LIN {X 0,Y 425.301,Z 259.752,A -85,B 0,C 180,E1 15177.061,E2 15177.061} C_VEL
LIN {X 0,Y 425.303,Z 259.751,A -85,B 0,C 180,E1 15173.169,E2 15173.169} C_VEL
LIN {X 0,Y 425.314,Z 259.743,A -85,B 0,C 180,E1 15169.371,E2 15169.371} C_VEL
LIN {X 0,Y 425.315,Z 259.738,A -85,B 0,C 180,E1 15165.531,E2 15165.531} C_VEL
LIN {X 0,Y 425.318,Z 259.739,A -85,B 0,C 180,E1 15161.623,E2 15161.623} C_VEL
LIN {X 0,Y 425.32,Z 259.754,A -85,B 0,C 180,E1 15157.829,E2 15157.829} C_VEL
LIN {X 0,Y 425.32,Z 259.751,A -85,B 0,C 180,E1 15153.921,E2 15153.921} C_VEL
LIN {X 0,Y 425.319,Z 259.736,A -85,B 0,C 180,E1 15150.046,E2 15150.046} C_VEL
LIN {X 0,Y 425.304,Z 259.744,A -85,B 0,C 180,E1 15146.228,E2 15146.228} C_VEL
LIN {X 0,Y 425.298,Z 259.757,A -85,B 0,C 180,E1 15142.385,E2 15142.385} C_VEL
LIN {X 0,Y 425.297,Z 259.743,A -85,B 0,C 180,E1 15138.503,E2 15138.503} C_VEL
LIN {X 0,Y 425.3,Z 259.734,A -85,B 0,C 180,E1 15134.707,E2 15134.707} C_VEL
LIN {X 0,Y 425.309,Z 259.756,A -85,B 0,C 180,E1 15130.839,E2 15130.839} C_VEL
LIN {X 0,Y 425.321,Z 259.742,A -85,B 0,C 180,E1 15127.02,E2 15127.02} C_VEL
LIN {X 0,Y 425.315,Z 259.735,A -85,B 0,C 180,E1 15123.098,E2 15123.098} C_VEL
LIN {X 0,Y 425.324,Z 259.753,A -85,B 0,C 180,E1 15119.325,E2 15119.325} C_VEL
LIN {X 0,Y 425.313,Z 259.752,A -85,B 0,C 180,E1 15115.414,E2 15115.414} C_VEL
LIN {X 0,Y 425.303,Z 259.742,A -85,B 0,C 180,E1 15111.618,E2 15111.618} C_VEL
LIN {X 0,Y 425.292,Z 259.736,A -85,B 0,C 180,E1 15107.784,E2 15107.784} C_VEL
LIN {X 0,Y 425.293,Z 259.748,A -85,B 0,C 180,E1 15104.033,E2 15104.033} C_VEL
LIN {X 0,Y 425.3,Z 259.753,A -85,B 0,C 180,E1 15100.211,E2 15100.211} C_VEL
LIN {X 0,Y 425.317,Z 259.755,A -85,B 0,C 180,E1 15096.443,E2 15096.443} C_VEL
LIN {X 0,Y 425.321,Z 259.752,A -85,B 0,C 180,E1 15092.563,E2 15092.563} C_VEL
LIN {X 0,Y 425.323,Z 259.747,A -85,B 0,C 180,E1 15088.698,E2 15088.698} C_VEL
LIN {X 0,Y 425.316,Z 259.743,A -85,B 0,C 180,E1 15084.832,E2 15084.832} C_VEL
LIN {X 0,Y 425.328,Z 259.912,A -85,B 0,C 180,E1 15083.057,E2 15083.057} C_VEL
LIN {X 0,Y 426.138,Z 262.4,A -85,B 0,C 180,E1 15082.576,E2 15082.576} C_VEL
LIN {X 0,Y 427.707,Z 264.913,A -85,B 0,C 180,E1 15082.061,E2 15082.061} C_VEL
LIN {X 0,Y 435.111,Z 279.75,A -85,B 0,C 180,E1 15079.434,E2 15079.434} C_VEL
LIN {X 0,Y 442.483,Z 295.067,A -85,B 0,C 180,E1 15076.967,E2 15076.967} C_VEL
LIN {X 0,Y 445.89,Z 302.403,A -85,B 0,C 180,E1 15075.916,E2 15075.916} C_VEL
LIN {X 0,Y 457.017,Z 320.95,A -85,B 0,C 180,E1 15074.239,E2 15074.239} C_VEL
LIN {X 0,Y 458.902,Z 336.106,A -85,B 0,C 180,E1 15073.722,E2 15073.722} C_VEL
LIN {X 0,Y 453.344,Z 551.105,A -85,B 0,C 180,E1 15070.004,E2 15070.004} C_VEL
LIN {X 0,Y 451.835,Z 606.521,A -85,B 0,C 180,E1 15069.024,E2 15069.024} C_VEL
LIN {X 0,Y 450.386,Z 628.482,A -85,B 0,C 180,E1 15068.425,E2 15068.425} C_VEL
LIN {X 0,Y 448.608,Z 649.294,A -85,B 0,C 180,E1 15067.637,E2 15067.637} C_VEL
LIN {X 0,Y 446.489,Z 669.88,A -85,B 0,C 180,E1 15066.638,E2 15066.638} C_VEL
LIN {X 0,Y 444.025,Z 690.18,A -85,B 0,C 180,E1 15065.397,E2 15065.397} C_VEL
LIN {X 0,Y 441.401,Z 709.749,A -85,B 0,C 180,E1 15063.941,E2 15063.941} C_VEL
LIN {X 0,Y 438.704,Z 728.638,A -85,B 0,C 180,E1 15062.268,E2 15062.268} C_VEL
LIN {X 0,Y 436.021,Z 746.682,A -85,B 0,C 180,E1 15060.372,E2 15060.372} C_VEL
LIN {X 0,Y 433.442,Z 763.445,A -85,B 0,C 180,E1 15058.295,E2 15058.295} C_VEL
LIN {X 0,Y 430.954,Z 780.217,A -85,B 0,C 180,E1 15055.858,E2 15055.858} C_VEL
LIN {X 0,Y 428.999,Z 794.198,A -85,B 0,C 180,E1 15053.485,E2 15053.485} C_VEL
LIN {X 0,Y 427.355,Z 806.771,A -85,B 0,C 180,E1 15050.974,E2 15050.974} C_VEL
LIN {X 0,Y 426.058,Z 818.033,A -85,B 0,C 180,E1 15048.327,E2 15048.327} C_VEL
LIN {X 0,Y 425.11,Z 827.973,A -85,B 0,C 180,E1 15045.551,E2 15045.551} C_VEL
LIN {X 0,Y 424.495,Z 835.991,A -85,B 0,C 180,E1 15042.79,E2 15042.79} C_VEL
LIN {X 0,Y 424.136,Z 842.606,A -85,B 0,C 180,E1 15039.908,E2 15039.908} C_VEL
LIN {X 0,Y 423.986,Z 847.351,A -85,B 0,C 180,E1 15037.178,E2 15037.178} C_VEL
LIN {X 0,Y 423.92,Z 850.446,A -85,B 0,C 180,E1 15034.463,E2 15034.463} C_VEL
LIN {X 0,Y 423.9,Z 852.175,A -85,B 0,C 180,E1 15031.756,E2 15031.756} C_VEL
LIN {X 0,Y 423.907,Z 852.32,A -85,B 0,C 180,E1 15029.053,E2 15029.053} C_VEL
LIN {X 0,Y 423.91,Z 851.039,A -85,B 0,C 180,E1 15026.212,E2 15026.212} C_VEL
LIN {X 0,Y 423.947,Z 848.381,A -85,B 0,C 180,E1 15023.634,E2 15023.634} C_VEL
LIN {X 0,Y 424.084,Z 843.921,A -85,B 0,C 180,E1 15020.773,E2 15020.773} C_VEL
LIN {X 0,Y 424.358,Z 838.352,A -85,B 0,C 180,E1 15018.17,E2 15018.17} C_VEL
LIN {X 0,Y 424.886,Z 830.435,A -85,B 0,C 180,E1 15015.276,E2 15015.276} C_VEL
LIN {X 0,Y 425.726,Z 821.114,A -85,B 0,C 180,E1 15012.504,E2 15012.504} C_VEL
LIN {X 0,Y 426.894,Z 810.324,A -85,B 0,C 180,E1 15009.86,E2 15009.86} C_VEL
LIN {X 0,Y 428.488,Z 797.377,A -85,B 0,C 180,E1 15007.179,E2 15007.179} C_VEL
LIN {X 0,Y 430.418,Z 783.285,A -85,B 0,C 180,E1 15004.694,E2 15004.694} C_VEL
LIN {X 0,Y 432.668,Z 767.834,A -85,B 0,C 180,E1 15002.369,E2 15002.369} C_VEL
LIN {X 0,Y 435.112,Z 751.206,A -85,B 0,C 180,E1 15000.24,E2 15000.24} C_VEL
LIN {X 0,Y 437.827,Z 732.887,A -85,B 0,C 180,E1 14998.237,E2 14998.237} C_VEL
LIN {X 0,Y 440.485,Z 714.446,A -85,B 0,C 180,E1 14996.523,E2 14996.523} C_VEL
LIN {X 0,Y 443.086,Z 695.133,A -85,B 0,C 180,E1 14995.027,E2 14995.027} C_VEL
LIN {X 0,Y 445.497,Z 675.185,A -85,B 0,C 180,E1 14993.743,E2 14993.743} C_VEL
LIN {X 0,Y 447.751,Z 654.688,A -85,B 0,C 180,E1 14992.67,E2 14992.67} C_VEL
LIN {X 0,Y 449.597,Z 634.166,A -85,B 0,C 180,E1 14991.836,E2 14991.836} C_VEL
LIN {X 0,Y 451.161,Z 611.946,A -85,B 0,C 180,E1 14991.172,E2 14991.172} C_VEL
LIN {X 0,Y 452.131,Z 587.924,A -85,B 0,C 180,E1 14990.684,E2 14990.684} C_VEL
LIN {X 0,Y 457.639,Z 367.78,A -85,B 0,C 180,E1 14986.894,E2 14986.894} C_VEL
LIN {X 0,Y 458.383,Z 333.61,A -85,B 0,C 180,E1 14986.271,E2 14986.271} C_VEL
LIN {X 0,Y 456.385,Z 319.925,A -85,B 0,C 180,E1 14985.758,E2 14985.758} C_VEL
LIN {X 0,Y 445.461,Z 301.473,A -85,B 0,C 180,E1 14984.048,E2 14984.048} C_VEL
LIN {X 0,Y 438.428,Z 285.88,A -85,B 0,C 180,E1 14981.579,E2 14981.579} C_VEL
LIN {X 0,Y 432.266,Z 273.434,A -85,B 0,C 180,E1 14979.33,E2 14979.33} C_VEL
LIN {X 0,Y 429.39,Z 268.237,A -85,B 0,C 180,E1 14978.273,E2 14978.273} C_VEL
LIN {X 0,Y 427.403,Z 264.222,A -85,B 0,C 180,E1 14977.463,E2 14977.463} C_VEL
LIN {X 0,Y 425.54,Z 260.917,A -85,B 0,C 180,E1 14976.726,E2 14976.726} C_VEL
LIN {X 0,Y 425.313,Z 259.812,A -85,B 0,C 180,E1 14976.395,E2 14976.395} C_VEL
LIN {X 0,Y 425.308,Z 259.758,A -85,B 0,C 180,E1 14972.573,E2 14972.573} C_VEL
LIN {X 0,Y 425.315,Z 259.748,A -85,B 0,C 180,E1 14968.731,E2 14968.731} C_VEL
LIN {X 0,Y 425.317,Z 259.757,A -85,B 0,C 180,E1 14964.846,E2 14964.846} C_VEL
LIN {X 0,Y 425.314,Z 259.749,A -85,B 0,C 180,E1 14961.043,E2 14961.043} C_VEL
LIN {X 0,Y 425.303,Z 259.747,A -85,B 0,C 180,E1 14957.231,E2 14957.231} C_VEL
LIN {X 0,Y 425.3,Z 259.753,A -85,B 0,C 180,E1 14953.46,E2 14953.46} C_VEL
LIN {X 0,Y 425.301,Z 259.76,A -85,B 0,C 180,E1 14949.61,E2 14949.61} C_VEL
LIN {X 0,Y 425.309,Z 259.756,A -85,B 0,C 180,E1 14945.803,E2 14945.803} C_VEL
LIN {X 0,Y 425.317,Z 259.749,A -85,B 0,C 180,E1 14942.022,E2 14942.022} C_VEL
LIN {X 0,Y 425.32,Z 259.746,A -85,B 0,C 180,E1 14938.25,E2 14938.25} C_VEL
LIN {X 0,Y 425.317,Z 259.756,A -85,B 0,C 180,E1 14934.335,E2 14934.335} C_VEL
LIN {X 0,Y 425.29,Z 259.754,A -85,B 0,C 180,E1 14930.666,E2 14930.666} C_VEL
LIN {X 0,Y 425.273,Z 259.761,A -85,B 0,C 180,E1 14926.957,E2 14926.957} C_VEL
LIN {X 0,Y 425.297,Z 259.923,A -85,B 0,C 180,E1 14924.805,E2 14924.805} C_VEL
LIN {X 0,Y 426.13,Z 262.406,A -85,B 0,C 180,E1 14924.207,E2 14924.207} C_VEL
LIN {X 0,Y 427.697,Z 265.015,A -85,B 0,C 180,E1 14923.57,E2 14923.57} C_VEL
LIN {X 0,Y 432.042,Z 273.926,A -85,B 0,C 180,E1 14921.656,E2 14921.656} C_VEL
LIN {X 0,Y 438.633,Z 288.164,A -85,B 0,C 180,E1 14918.892,E2 14918.892} C_VEL
LIN {X 0,Y 443.787,Z 300.497,A -85,B 0,C 180,E1 14916.798,E2 14916.798} C_VEL
LIN {X 0,Y 453.343,Z 316.481,A -85,B 0,C 180,E1 14915.244,E2 14915.244} C_VEL
LIN {X 0,Y 455.959,Z 333.247,A -85,B 0,C 180,E1 14914.568,E2 14914.568} C_VEL
LIN {X 0,Y 448.532,Z 567.509,A -85,B 0,C 180,E1 14910.326,E2 14910.326} C_VEL
LIN {X 0,Y 447.276,Z 588.491,A -85,B 0,C 180,E1 14909.711,E2 14909.711} C_VEL
LIN {X 0,Y 445.669,Z 608.284,A -85,B 0,C 180,E1 14908.896,E2 14908.896} C_VEL
LIN {X 0,Y 443.645,Z 628.289,A -85,B 0,C 180,E1 14907.823,E2 14907.823} C_VEL
LIN {X 0,Y 441.394,Z 647.121,A -85,B 0,C 180,E1 14906.553,E2 14906.553} C_VEL
LIN {X 0,Y 439.116,Z 664.26,A -85,B 0,C 180,E1 14905.146,E2 14905.146} C_VEL
LIN {X 0,Y 436.553,Z 681.806,A -85,B 0,C 180,E1 14903.408,E2 14903.408} C_VEL
LIN {X 0,Y 434.022,Z 698.14,A -85,B 0,C 180,E1 14901.455,E2 14901.455} C_VEL
LIN {X 0,Y 431.753,Z 712.503,A -85,B 0,C 180,E1 14899.405,E2 14899.405} C_VEL
LIN {X 0,Y 429.664,Z 725.853,A -85,B 0,C 180,E1 14897.142,E2 14897.142} C_VEL
LIN {X 0,Y 427.831,Z 738.286,A -85,B 0,C 180,E1 14894.611,E2 14894.611} C_VEL
LIN {X 0,Y 427.439,Z 741.15,A -85,B 0,C 180,E1 14893.967,E2 14893.967} C_VEL
LIN {X 0,Y 425.985,Z 745.086,A -85,B 0,C 180,E1 14893.089,E2 14893.089} C_VEL
LIN {X 0,Y 419.031,Z 754.446,A -85,B 0,C 180,E1 14890.859,E2 14890.859} C_VEL
LIN {X 0,Y 417.682,Z 757.489,A -85,B 0,C 180,E1 14889.897,E2 14889.897} C_VEL
LIN {X 0,Y 416.881,Z 764.999,A -85,B 0,C 180,E1 14886.999,E2 14886.999} C_VEL
LIN {X 0,Y 416.439,Z 770.435,A -85,B 0,C 180,E1 14884.184,E2 14884.184} C_VEL
LIN {X 0,Y 416.212,Z 774.156,A -85,B 0,C 180,E1 14881.42,E2 14881.42} C_VEL
LIN {X 0,Y 416.135,Z 776.403,A -85,B 0,C 180,E1 14878.565,E2 14878.565} C_VEL
LIN {X 0,Y 416.109,Z 777.068,A -85,B 0,C 180,E1 14875.782,E2 14875.782} C_VEL
LIN {X 0,Y 416.131,Z 776.179,A -85,B 0,C 180,E1 14873.042,E2 14873.042} C_VEL
LIN {X 0,Y 416.214,Z 773.712,A -85,B 0,C 180,E1 14870.24,E2 14870.24} C_VEL
LIN {X 0,Y 416.448,Z 769.461,A -85,B 0,C 180,E1 14867.322,E2 14867.322} C_VEL
LIN {X 0,Y 416.897,Z 763.841,A -85,B 0,C 180,E1 14864.587,E2 14864.587} C_VEL
LIN {X 0,Y 417.65,Z 756.615,A -85,B 0,C 180,E1 14861.883,E2 14861.883} C_VEL
LIN {X 0,Y 418.842,Z 747.081,A -85,B 0,C 180,E1 14859.066,E2 14859.066} C_VEL
LIN {X 0,Y 420.424,Z 735.997,A -85,B 0,C 180,E1 14856.419,E2 14856.419} C_VEL
LIN {X 0,Y 422.248,Z 724.149,A -85,B 0,C 180,E1 14854.075,E2 14854.075} C_VEL
LIN {X 0,Y 424.353,Z 711.065,A -85,B 0,C 180,E1 14851.892,E2 14851.892} C_VEL
LIN {X 0,Y 426.769,Z 696.203,A -85,B 0,C 180,E1 14849.8,E2 14849.8} C_VEL
LIN {X 0,Y 429.265,Z 680.441,A -85,B 0,C 180,E1 14847.932,E2 14847.932} C_VEL
LIN {X 0,Y 431.865,Z 663.081,A -85,B 0,C 180,E1 14846.217,E2 14846.217} C_VEL
LIN {X 0,Y 434.365,Z 644.633,A -85,B 0,C 180,E1 14844.718,E2 14844.718} C_VEL
LIN {X 0,Y 436.594,Z 626.086,A -85,B 0,C 180,E1 14843.492,E2 14843.492} C_VEL
LIN {X 0,Y 438.597,Z 606.057,A -85,B 0,C 180,E1 14842.436,E2 14842.436} C_VEL
LIN {X 0,Y 440.289,Z 585.271,A -85,B 0,C 180,E1 14841.612,E2 14841.612} C_VEL
LIN {X 0,Y 441.466,Z 564.974,A -85,B 0,C 180,E1 14841.039,E2 14841.039} C_VEL
LIN {X 0,Y 448.439,Z 333.3,A -85,B 0,C 180,E1 14836.885,E2 14836.885} C_VEL
LIN {X 0,Y 445.796,Z 318.48,A -85,B 0,C 180,E1 14836.272,E2 14836.272} C_VEL
LIN {X 0,Y 434.687,Z 299.71,A -85,B 0,C 180,E1 14834.524,E2 14834.524} C_VEL
LIN {X 0,Y 427.785,Z 283.545,A -85,B 0,C 180,E1 14831.75,E2 14831.75} C_VEL
LIN {X 0,Y 422.474,Z 272.072,A -85,B 0,C 180,E1 14829.581,E2 14829.581} C_VEL
LIN {X 0,Y 419.084,Z 264.754,A -85,B 0,C 180,E1 14828.133,E2 14828.133} C_VEL
LIN {X 0,Y 417.393,Z 260.937,A -85,B 0,C 180,E1 14827.316,E2 14827.316} C_VEL
LIN {X 0,Y 417.378,Z 260.734,A -85,B 0,C 180,E1 14823.848,E2 14823.848} C_VEL
LIN {X 0,Y 417.382,Z 260.747,A -85,B 0,C 180,E1 14819.958,E2 14819.958} C_VEL
LIN {X 0,Y 417.38,Z 260.747,A -85,B 0,C 180,E1 14815.979,E2 14815.979} C_VEL
LIN {X 0,Y 417.382,Z 260.746,A -85,B 0,C 180,E1 14812.003,E2 14812.003} C_VEL
LIN {X 0,Y 417.381,Z 260.744,A -85,B 0,C 180,E1 14808.062,E2 14808.062} C_VEL
LIN {X 0,Y 417.379,Z 260.74,A -85,B 0,C 180,E1 14804.193,E2 14804.193} C_VEL
LIN {X 0,Y 417.374,Z 260.727,A -85,B 0,C 180,E1 14800.299,E2 14800.299} C_VEL
LIN {X 0,Y 417.362,Z 260.725,A -85,B 0,C 180,E1 14796.448,E2 14796.448} C_VEL
LIN {X 0,Y 417.36,Z 260.741,A -85,B 0,C 180,E1 14792.615,E2 14792.615} C_VEL
LIN {X 0,Y 417.362,Z 260.745,A -85,B 0,C 180,E1 14788.744,E2 14788.744} C_VEL
LIN {X 0,Y 417.366,Z 260.724,A -85,B 0,C 180,E1 14784.936,E2 14784.936} C_VEL
LIN {X 0,Y 417.376,Z 260.733,A -85,B 0,C 180,E1 14781.058,E2 14781.058} C_VEL
LIN {X 0,Y 417.377,Z 260.744,A -85,B 0,C 180,E1 14777.099,E2 14777.099} C_VEL
LIN {X 0,Y 417.379,Z 260.719,A -85,B 0,C 180,E1 14773.294,E2 14773.294} C_VEL
LIN {X 0,Y 417.379,Z 260.728,A -85,B 0,C 180,E1 14769.374,E2 14769.374} C_VEL
LIN {X 0,Y 417.379,Z 260.744,A -85,B 0,C 180,E1 14765.497,E2 14765.497} C_VEL
LIN {X 0,Y 417.372,Z 260.734,A -85,B 0,C 180,E1 14761.646,E2 14761.646} C_VEL
LIN {X 0,Y 417.355,Z 260.724,A -85,B 0,C 180,E1 14757.94,E2 14757.94} C_VEL
LIN {X 0,Y 417.353,Z 260.741,A -85,B 0,C 180,E1 14754.086,E2 14754.086} C_VEL
LIN {X 0,Y 417.357,Z 260.747,A -85,B 0,C 180,E1 14750.206,E2 14750.206} C_VEL
LIN {X 0,Y 417.368,Z 260.733,A -85,B 0,C 180,E1 14746.421,E2 14746.421} C_VEL
LIN {X 0,Y 417.374,Z 260.728,A -85,B 0,C 180,E1 14742.575,E2 14742.575} C_VEL
LIN {X 0,Y 417.384,Z 260.727,A -85,B 0,C 180,E1 14738.646,E2 14738.646} C_VEL
LIN {X 0,Y 417.38,Z 260.729,A -85,B 0,C 180,E1 14734.759,E2 14734.759} C_VEL
LIN {X 0,Y 417.382,Z 260.729,A -85,B 0,C 180,E1 14730.902,E2 14730.902} C_VEL
LIN {X 0,Y 417.371,Z 260.738,A -85,B 0,C 180,E1 14727.056,E2 14727.056} C_VEL
LIN {X 0,Y 417.408,Z 261.004,A -85,B 0,C 180,E1 14724.197,E2 14724.197} C_VEL
LIN {X 0,Y 418.758,Z 264.378,A -85,B 0,C 180,E1 14723.52,E2 14723.52} C_VEL
LIN {X 0,Y 419.926,Z 266.204,A -85,B 0,C 180,E1 14723.128,E2 14723.128} C_VEL
LIN {X 0,Y 426.82,Z 279.835,A -85,B 0,C 180,E1 14720.591,E2 14720.591} C_VEL
LIN {X 0,Y 434.436,Z 295.417,A -85,B 0,C 180,E1 14717.952,E2 14717.952} C_VEL
LIN {X 0,Y 437.761,Z 302.391,A -85,B 0,C 180,E1 14716.904,E2 14716.904} C_VEL
LIN {X 0,Y 450.827,Z 323.776,A -85,B 0,C 180,E1 14714.879,E2 14714.879} C_VEL
LIN {X 0,Y 451.465,Z 325.832,A -85,B 0,C 180,E1 14714.762,E2 14714.762} C_VEL
LIN {X 0,Y 452.833,Z 337.546,A -85,B 0,C 180,E1 14714.362,E2 14714.362} C_VEL
LIN {X 0,Y 446.973,Z 551.29,A -85,B 0,C 180,E1 14710.621,E2 14710.621} C_VEL
LIN {X 0,Y 445.404,Z 606.186,A -85,B 0,C 180,E1 14709.639,E2 14709.639} C_VEL
LIN {X 0,Y 443.876,Z 628.267,A -85,B 0,C 180,E1 14709.032,E2 14709.032} C_VEL
LIN {X 0,Y 441.975,Z 649.397,A -85,B 0,C 180,E1 14708.221,E2 14708.221} C_VEL
LIN {X 0,Y 439.756,Z 669.844,A -85,B 0,C 180,E1 14707.212,E2 14707.212} C_VEL
LIN {X 0,Y 437.228,Z 689.56,A -85,B 0,C 180,E1 14705.992,E2 14705.992} C_VEL
LIN {X 0,Y 434.471,Z 709.083,A -85,B 0,C 180,E1 14704.525,E2 14704.525} C_VEL
LIN {X 0,Y 431.62,Z 728.067,A -85,B 0,C 180,E1 14702.822,E2 14702.822} C_VEL
LIN {X 0,Y 428.809,Z 745.853,A -85,B 0,C 180,E1 14700.93,E2 14700.93} C_VEL
LIN {X 0,Y 426.062,Z 762.77,A -85,B 0,C 180,E1 14698.806,E2 14698.806} C_VEL
LIN {X 0,Y 423.441,Z 779.408,A -85,B 0,C 180,E1 14696.352,E2 14696.352} C_VEL
LIN {X 0,Y 421.351,Z 793.415,A -85,B 0,C 180,E1 14693.938,E2 14693.938} C_VEL
LIN {X 0,Y 419.527,Z 806.506,A -85,B 0,C 180,E1 14691.271,E2 14691.271} C_VEL
LIN {X 0,Y 418.14,Z 817.819,A -85,B 0,C 180,E1 14688.542,E2 14688.542} C_VEL
LIN {X 0,Y 417.148,Z 827.661,A -85,B 0,C 180,E1 14685.713,E2 14685.713} C_VEL
LIN {X 0,Y 416.521,Z 835.522,A -85,B 0,C 180,E1 14682.939,E2 14682.939} C_VEL
LIN {X 0,Y 416.161,Z 841.887,A -85,B 0,C 180,E1 14680.1,E2 14680.1} C_VEL
LIN {X 0,Y 416.001,Z 846.635,A -85,B 0,C 180,E1 14677.317,E2 14677.317} C_VEL
LIN {X 0,Y 415.946,Z 849.737,A -85,B 0,C 180,E1 14674.548,E2 14674.548} C_VEL
LIN {X 0,Y 415.929,Z 851.481,A -85,B 0,C 180,E1 14671.789,E2 14671.789} C_VEL
LIN {X 0,Y 415.938,Z 851.63,A -85,B 0,C 180,E1 14669.034,E2 14669.034} C_VEL
LIN {X 0,Y 415.938,Z 850.315,A -85,B 0,C 180,E1 14666.139,E2 14666.139} C_VEL
LIN {X 0,Y 415.97,Z 847.646,A -85,B 0,C 180,E1 14663.512,E2 14663.512} C_VEL
LIN {X 0,Y 416.112,Z 843.169,A -85,B 0,C 180,E1 14660.595,E2 14660.595} C_VEL
LIN {X 0,Y 416.393,Z 837.583,A -85,B 0,C 180,E1 14657.94,E2 14657.94} C_VEL
LIN {X 0,Y 416.955,Z 829.643,A -85,B 0,C 180,E1 14654.989,E2 14654.989} C_VEL
LIN {X 0,Y 417.85,Z 820.294,A -85,B 0,C 180,E1 14652.163,E2 14652.163} C_VEL
LIN {X 0,Y 419.089,Z 809.483,A -85,B 0,C 180,E1 14649.468,E2 14649.468} C_VEL
LIN {X 0,Y 420.774,Z 796.654,A -85,B 0,C 180,E1 14646.767,E2 14646.767} C_VEL
LIN {X 0,Y 422.773,Z 782.932,A -85,B 0,C 180,E1 14644.299,E2 14644.299} C_VEL
LIN {X 0,Y 425.145,Z 767.555,A -85,B 0,C 180,E1 14641.941,E2 14641.941} C_VEL
LIN {X 0,Y 427.673,Z 751.38,A -85,B 0,C 180,E1 14639.823,E2 14639.823} C_VEL
LIN {X 0,Y 430.524,Z 733.225,A -85,B 0,C 180,E1 14637.791,E2 14637.791} C_VEL
LIN {X 0,Y 433.317,Z 714.948,A -85,B 0,C 180,E1 14636.053,E2 14636.053} C_VEL
LIN {X 0,Y 436.043,Z 695.823,A -85,B 0,C 180,E1 14634.539,E2 14634.539} C_VEL
LIN {X 0,Y 438.714,Z 675.069,A -85,B 0,C 180,E1 14633.172,E2 14633.172} C_VEL
LIN {X 0,Y 441.125,Z 654.322,A -85,B 0,C 180,E1 14632.072,E2 14632.072} C_VEL
LIN {X 0,Y 443.069,Z 633.728,A -85,B 0,C 180,E1 14631.227,E2 14631.227} C_VEL
LIN {X 0,Y 444.705,Z 611.527,A -85,B 0,C 180,E1 14630.556,E2 14630.556} C_VEL
LIN {X 0,Y 445.729,Z 587.428,A -85,B 0,C 180,E1 14630.062,E2 14630.062} C_VEL
LIN {X 0,Y 451.614,Z 367.128,A -85,B 0,C 180,E1 14626.218,E2 14626.218} C_VEL
LIN {X 0,Y 452.376,Z 335.05,A -85,B 0,C 180,E1 14625.623,E2 14625.623} C_VEL
LIN {X 0,Y 450.779,Z 323.87,A -85,B 0,C 180,E1 14625.195,E2 14625.195} C_VEL
LIN {X 0,Y 439.766,Z 305.361,A -85,B 0,C 180,E1 14623.432,E2 14623.432} C_VEL
LIN {X 0,Y 437.248,Z 301.106,A -85,B 0,C 180,E1 14622.957,E2 14622.957} C_VEL
LIN {X 0,Y 430.638,Z 286.826,A -85,B 0,C 180,E1 14620.55,E2 14620.55} C_VEL
LIN {X 0,Y 424.299,Z 274.319,A -85,B 0,C 180,E1 14618.127,E2 14618.127} C_VEL
LIN {X 0,Y 421.933,Z 269.831,A -85,B 0,C 180,E1 14617.177,E2 14617.177} C_VEL
LIN {X 0,Y 419.29,Z 265.018,A -85,B 0,C 180,E1 14616.087,E2 14616.087} C_VEL
LIN {X 0,Y 417.597,Z 261.86,A -85,B 0,C 180,E1 14615.349,E2 14615.349} C_VEL
LIN {X 0,Y 417.383,Z 260.784,A -85,B 0,C 180,E1 14614.986,E2 14614.986} C_VEL
LIN {X 0,Y 417.38,Z 260.739,A -85,B 0,C 180,E1 14611.161,E2 14611.161} C_VEL
LIN {X 0,Y 417.376,Z 260.742,A -85,B 0,C 180,E1 14607.23,E2 14607.23} C_VEL
LIN {X 0,Y 417.37,Z 260.736,A -85,B 0,C 180,E1 14603.431,E2 14603.431} C_VEL
LIN {X 0,Y 417.369,Z 260.742,A -85,B 0,C 180,E1 14599.597,E2 14599.597} C_VEL
LIN {X 0,Y 417.37,Z 260.747,A -85,B 0,C 180,E1 14595.707,E2 14595.707} C_VEL
LIN {X 0,Y 417.373,Z 260.739,A -85,B 0,C 180,E1 14591.89,E2 14591.89} C_VEL
LIN {X 0,Y 417.382,Z 260.734,A -85,B 0,C 180,E1 14587.988,E2 14587.988} C_VEL
LIN {X 0,Y 417.377,Z 260.735,A -85,B 0,C 180,E1 14584.122,E2 14584.122} C_VEL
LIN {X 0,Y 417.386,Z 260.742,A -85,B 0,C 180,E1 14580.276,E2 14580.276} C_VEL
LIN {X 0,Y 417.373,Z 260.743,A -85,B 0,C 180,E1 14576.43,E2 14576.43} C_VEL
LIN {X 0,Y 417.36,Z 260.738,A -85,B 0,C 180,E1 14572.568,E2 14572.568} C_VEL
LIN {X 0,Y 417.343,Z 260.75,A -85,B 0,C 180,E1 14568.812,E2 14568.812} C_VEL
LIN {X 0,Y 417.418,Z 261.002,A -85,B 0,C 180,E1 14566.142,E2 14566.142} C_VEL
LIN {X 0,Y 419.005,Z 264.731,A -85,B 0,C 180,E1 14565.208,E2 14565.208} C_VEL
LIN {X 0,Y 419.923,Z 266.22,A -85,B 0,C 180,E1 14564.818,E2 14564.818} C_VEL
LIN {X 0,Y 422.649,Z 271.937,A -85,B 0,C 180,E1 14563.509,E2 14563.509} C_VEL
LIN {X 0,Y 426.19,Z 278.883,A -85,B 0,C 180,E1 14561.962,E2 14561.962} C_VEL
LIN {X 0,Y 432.656,Z 293.106,A -85,B 0,C 180,E1 14559.153,E2 14559.153} C_VEL
LIN {X 0,Y 435.89,Z 300.619,A -85,B 0,C 180,E1 14557.851,E2 14557.851} C_VEL
LIN {X 0,Y 446.307,Z 317.854,A -85,B 0,C 180,E1 14556.064,E2 14556.064} C_VEL
LIN {X 0,Y 447.954,Z 321.052,A -85,B 0,C 180,E1 14555.788,E2 14555.788} C_VEL
LIN {X 0,Y 450.008,Z 334.928,A -85,B 0,C 180,E1 14555.226,E2 14555.226} C_VEL
LIN {X 0,Y 442.171,Z 567.894,A -85,B 0,C 180,E1 14550.949,E2 14550.949} C_VEL
LIN {X 0,Y 440.859,Z 588.788,A -85,B 0,C 180,E1 14550.329,E2 14550.329} C_VEL
LIN {X 0,Y 439.239,Z 607.795,A -85,B 0,C 180,E1 14549.544,E2 14549.544} C_VEL
LIN {X 0,Y 437.088,Z 628.269,A -85,B 0,C 180,E1 14548.443,E2 14548.443} C_VEL
LIN {X 0,Y 434.784,Z 646.724,A -85,B 0,C 180,E1 14547.197,E2 14547.197} C_VEL
LIN {X 0,Y 432.374,Z 664.01,A -85,B 0,C 180,E1 14545.776,E2 14545.776} C_VEL
LIN {X 0,Y 429.72,Z 681.134,A -85,B 0,C 180,E1 14544.07,E2 14544.07} C_VEL
LIN {X 0,Y 427.258,Z 696.202,A -85,B 0,C 180,E1 14542.279,E2 14542.279} C_VEL
LIN {X 0,Y 424.701,Z 711.448,A -85,B 0,C 180,E1 14540.13,E2 14540.13} C_VEL
LIN {X 0,Y 422.406,Z 725.223,A -85,B 0,C 180,E1 14537.809,E2 14537.809} C_VEL
LIN {X 0,Y 420.548,Z 736.884,A -85,B 0,C 180,E1 14535.466,E2 14535.466} C_VEL
LIN {X 0,Y 418.957,Z 747.652,A -85,B 0,C 180,E1 14532.858,E2 14532.858} C_VEL
LIN {X 0,Y 417.72,Z 757.152,A -85,B 0,C 180,E1 14530.011,E2 14530.011} C_VEL
LIN {X 0,Y 417.682,Z 757.489,A -85,B 0,C 180,E1 14529.897,E2 14529.897} C_VEL
LIN {X 0,Y 416.383,Z 760.385,A -85,B 0,C 180,E1 14528.921,E2 14528.921} C_VEL
LIN {X 0,Y 409.57,Z 767.591,A -85,B 0,C 180,E1 14526.311,E2 14526.311} C_VEL
LIN {X 0,Y 408.663,Z 769.356,A -85,B 0,C 180,E1 14525.419,E2 14525.419} C_VEL
LIN {X 0,Y 408.332,Z 773.921,A -85,B 0,C 180,E1 14522.43,E2 14522.43} C_VEL
LIN {X 0,Y 408.193,Z 776.567,A -85,B 0,C 180,E1 14519.596,E2 14519.596} C_VEL
LIN {X 0,Y 408.146,Z 777.699,A -85,B 0,C 180,E1 14516.793,E2 14516.793} C_VEL
LIN {X 0,Y 408.152,Z 777.365,A -85,B 0,C 180,E1 14513.977,E2 14513.977} C_VEL
LIN {X 0,Y 408.23,Z 775.454,A -85,B 0,C 180,E1 14511.072,E2 14511.072} C_VEL
LIN {X 0,Y 408.405,Z 771.914,A -85,B 0,C 180,E1 14508.219,E2 14508.219} C_VEL
LIN {X 0,Y 408.792,Z 766.942,A -85,B 0,C 180,E1 14505.463,E2 14505.463} C_VEL
LIN {X 0,Y 409.518,Z 759.939,A -85,B 0,C 180,E1 14502.552,E2 14502.552} C_VEL
LIN {X 0,Y 410.58,Z 751.56,A -85,B 0,C 180,E1 14499.816,E2 14499.816} C_VEL
LIN {X 0,Y 412.002,Z 741.93,A -85,B 0,C 180,E1 14497.251,E2 14497.251} C_VEL
LIN {X 0,Y 413.975,Z 729.658,A -85,B 0,C 180,E1 14494.573,E2 14494.573} C_VEL
LIN {X 0,Y 416.225,Z 716.34,A -85,B 0,C 180,E1 14492.172,E2 14492.172} C_VEL
LIN {X 0,Y 418.676,Z 701.979,A -85,B 0,C 180,E1 14490.001,E2 14490.001} C_VEL
LIN {X 0,Y 421.306,Z 686.455,A -85,B 0,C 180,E1 14488.029,E2 14488.029} C_VEL
LIN {X 0,Y 424.044,Z 669.404,A -85,B 0,C 180,E1 14486.216,E2 14486.216} C_VEL
LIN {X 0,Y 426.617,Z 652.172,A -85,B 0,C 180,E1 14484.69,E2 14484.69} C_VEL
LIN {X 0,Y 429.148,Z 633.198,A -85,B 0,C 180,E1 14483.312,E2 14483.312} C_VEL
LIN {X 0,Y 431.302,Z 614.093,A -85,B 0,C 180,E1 14482.207,E2 14482.207} C_VEL
LIN {X 0,Y 433.132,Z 594.076,A -85,B 0,C 180,E1 14481.305,E2 14481.305} C_VEL
LIN {X 0,Y 434.615,Z 572.841,A -85,B 0,C 180,E1 14480.61,E2 14480.61} C_VEL
LIN {X 0,Y 435.638,Z 548.232,A -85,B 0,C 180,E1 14480.085,E2 14480.085} C_VEL
LIN {X 0,Y 442.318,Z 334.616,A -85,B 0,C 180,E1 14476.225,E2 14476.225} C_VEL
LIN {X 0,Y 440.136,Z 322.454,A -85,B 0,C 180,E1 14475.707,E2 14475.707} C_VEL
LIN {X 0,Y 428.487,Z 302.94,A -85,B 0,C 180,E1 14473.837,E2 14473.837} C_VEL
LIN {X 0,Y 426.191,Z 298.916,A -85,B 0,C 180,E1 14473.37,E2 14473.37} C_VEL
LIN {X 0,Y 418.994,Z 282.204,A -85,B 0,C 180,E1 14470.34,E2 14470.34} C_VEL
LIN {X 0,Y 412.758,Z 269.25,A -85,B 0,C 180,E1 14467.716,E2 14467.716} C_VEL
LIN {X 0,Y 410.89,Z 265.39,A -85,B 0,C 180,E1 14466.895,E2 14466.895} C_VEL
LIN {X 0,Y 409.472,Z 261.946,A -85,B 0,C 180,E1 14466.128,E2 14466.128} C_VEL
LIN {X 0,Y 409.427,Z 261.737,A -85,B 0,C 180,E1 14462.987,E2 14462.987} C_VEL
LIN {X 0,Y 409.426,Z 261.729,A -85,B 0,C 180,E1 14459.149,E2 14459.149} C_VEL
LIN {X 0,Y 409.428,Z 261.726,A -85,B 0,C 180,E1 14455.321,E2 14455.321} C_VEL
LIN {X 0,Y 409.434,Z 261.726,A -85,B 0,C 180,E1 14451.391,E2 14451.391} C_VEL
LIN {X 0,Y 409.437,Z 261.731,A -85,B 0,C 180,E1 14447.436,E2 14447.436} C_VEL
LIN {X 0,Y 409.44,Z 261.735,A -85,B 0,C 180,E1 14443.511,E2 14443.511} C_VEL
LIN {X 0,Y 409.442,Z 261.722,A -85,B 0,C 180,E1 14439.593,E2 14439.593} C_VEL
LIN {X 0,Y 409.437,Z 261.709,A -85,B 0,C 180,E1 14435.705,E2 14435.705} C_VEL
LIN {X 0,Y 409.44,Z 261.718,A -85,B 0,C 180,E1 14431.812,E2 14431.812} C_VEL
LIN {X 0,Y 409.448,Z 261.732,A -85,B 0,C 180,E1 14427.877,E2 14427.877} C_VEL
LIN {X 0,Y 409.437,Z 261.722,A -85,B 0,C 180,E1 14423.913,E2 14423.913} C_VEL
LIN {X 0,Y 409.426,Z 261.712,A -85,B 0,C 180,E1 14420.14,E2 14420.14} C_VEL
LIN {X 0,Y 409.419,Z 261.732,A -85,B 0,C 180,E1 14416.309,E2 14416.309} C_VEL
LIN {X 0,Y 409.419,Z 261.727,A -85,B 0,C 180,E1 14412.361,E2 14412.361} C_VEL
LIN {X 0,Y 409.416,Z 261.711,A -85,B 0,C 180,E1 14408.425,E2 14408.425} C_VEL
LIN {X 0,Y 409.426,Z 261.728,A -85,B 0,C 180,E1 14404.621,E2 14404.621} C_VEL
LIN {X 0,Y 409.434,Z 261.732,A -85,B 0,C 180,E1 14400.698,E2 14400.698} C_VEL
LIN {X 0,Y 409.433,Z 261.712,A -85,B 0,C 180,E1 14396.779,E2 14396.779} C_VEL
LIN {X 0,Y 409.445,Z 261.711,A -85,B 0,C 180,E1 14392.845,E2 14392.845} C_VEL
LIN {X 0,Y 409.44,Z 261.721,A -85,B 0,C 180,E1 14388.876,E2 14388.876} C_VEL
LIN {X 0,Y 409.448,Z 261.734,A -85,B 0,C 180,E1 14384.997,E2 14384.997} C_VEL
LIN {X 0,Y 409.441,Z 261.733,A -85,B 0,C 180,E1 14381.046,E2 14381.046} C_VEL
LIN {X 0,Y 409.44,Z 261.733,A -85,B 0,C 180,E1 14377.152,E2 14377.152} C_VEL
LIN {X 0,Y 409.426,Z 261.736,A -85,B 0,C 180,E1 14373.297,E2 14373.297} C_VEL
LIN {X 0,Y 409.418,Z 261.738,A -85,B 0,C 180,E1 14369.471,E2 14369.471} C_VEL
LIN {X 0,Y 409.424,Z 261.808,A -85,B 0,C 180,E1 14365.53,E2 14365.53} C_VEL
LIN {X 0,Y 409.727,Z 263.117,A -85,B 0,C 180,E1 14365.177,E2 14365.177} C_VEL
LIN {X 0,Y 412.155,Z 267.655,A -85,B 0,C 180,E1 14364.221,E2 14364.221} C_VEL
LIN {X 0,Y 416.793,Z 276.512,A -85,B 0,C 180,E1 14362.458,E2 14362.458} C_VEL
LIN {X 0,Y 423.779,Z 290.492,A -85,B 0,C 180,E1 14359.9,E2 14359.9} C_VEL
LIN {X 0,Y 429.505,Z 302.322,A -85,B 0,C 180,E1 14357.965,E2 14357.965} C_VEL
LIN {X 0,Y 443.428,Z 324.749,A -85,B 0,C 180,E1 14355.72,E2 14355.72} C_VEL
LIN {X 0,Y 445.708,Z 329.008,A -85,B 0,C 180,E1 14355.36,E2 14355.36} C_VEL
LIN {X 0,Y 446.813,Z 338.96,A -85,B 0,C 180,E1 14355.017,E2 14355.017} C_VEL
LIN {X 0,Y 440.618,Z 552.594,A -85,B 0,C 180,E1 14351.234,E2 14351.234} C_VEL
LIN {X 0,Y 439.011,Z 605.794,A -85,B 0,C 180,E1 14350.27,E2 14350.27} C_VEL
LIN {X 0,Y 437.412,Z 627.846,A -85,B 0,C 180,E1 14349.66,E2 14349.66} C_VEL
LIN {X 0,Y 435.474,Z 648.473,A -85,B 0,C 180,E1 14348.864,E2 14348.864} C_VEL
LIN {X 0,Y 433.225,Z 668.6,A -85,B 0,C 180,E1 14347.871,E2 14347.871} C_VEL
LIN {X 0,Y 430.556,Z 688.426,A -85,B 0,C 180,E1 14346.64,E2 14346.64} C_VEL
LIN {X 0,Y 427.57,Z 708.552,A -85,B 0,C 180,E1 14345.116,E2 14345.116} C_VEL
LIN {X 0,Y 424.644,Z 727.13,A -85,B 0,C 180,E1 14343.432,E2 14343.432} C_VEL
LIN {X 0,Y 421.668,Z 744.785,A -85,B 0,C 180,E1 14341.533,E2 14341.533} C_VEL
LIN {X 0,Y 418.874,Z 761.225,A -85,B 0,C 180,E1 14339.452,E2 14339.452} C_VEL
LIN {X 0,Y 416.254,Z 776.845,A -85,B 0,C 180,E1 14337.152,E2 14337.152} C_VEL
LIN {X 0,Y 413.952,Z 791.067,A -85,B 0,C 180,E1 14334.698,E2 14334.698} C_VEL
LIN {X 0,Y 412.021,Z 803.901,A -85,B 0,C 180,E1 14332.093,E2 14332.093} C_VEL
LIN {X 0,Y 410.497,Z 815.45,A -85,B 0,C 180,E1 14329.343,E2 14329.343} C_VEL
LIN {X 0,Y 409.415,Z 825.111,A -85,B 0,C 180,E1 14326.601,E2 14326.601} C_VEL
LIN {X 0,Y 408.665,Z 833.416,A -85,B 0,C 180,E1 14323.727,E2 14323.727} C_VEL
LIN {X 0,Y 408.243,Z 840.126,A -85,B 0,C 180,E1 14320.85,E2 14320.85} C_VEL
LIN {X 0,Y 408.045,Z 845.05,A -85,B 0,C 180,E1 14318.027,E2 14318.027} C_VEL
LIN {X 0,Y 407.979,Z 848.664,A -85,B 0,C 180,E1 14315.06,E2 14315.06} C_VEL
LIN {X 0,Y 407.966,Z 850.498,A -85,B 0,C 180,E1 14312.386,E2 14312.386} C_VEL
LIN {X 0,Y 407.961,Z 850.986,A -85,B 0,C 180,E1 14309.437,E2 14309.437} C_VEL
LIN {X 0,Y 407.972,Z 850.041,A -85,B 0,C 180,E1 14306.767,E2 14306.767} C_VEL
LIN {X 0,Y 407.988,Z 847.42,A -85,B 0,C 180,E1 14303.808,E2 14303.808} C_VEL
LIN {X 0,Y 408.089,Z 843.433,A -85,B 0,C 180,E1 14300.977,E2 14300.977} C_VEL
LIN {X 0,Y 408.37,Z 837.781,A -85,B 0,C 180,E1 14298.13,E2 14298.13} C_VEL
LIN {X 0,Y 408.88,Z 830.563,A -85,B 0,C 180,E1 14295.266,E2 14295.266} C_VEL
LIN {X 0,Y 409.701,Z 821.968,A -85,B 0,C 180,E1 14292.53,E2 14292.53} C_VEL
LIN {X 0,Y 410.991,Z 811.058,A -85,B 0,C 180,E1 14289.64,E2 14289.64} C_VEL
LIN {X 0,Y 412.588,Z 799.452,A -85,B 0,C 180,E1 14287.034,E2 14287.034} C_VEL
LIN {X 0,Y 414.692,Z 785.455,A -85,B 0,C 180,E1 14284.389,E2 14284.389} C_VEL
LIN {X 0,Y 417.104,Z 770.491,A -85,B 0,C 180,E1 14281.975,E2 14281.975} C_VEL
LIN {X 0,Y 419.78,Z 754.44,A -85,B 0,C 180,E1 14279.749,E2 14279.749} C_VEL
LIN {X 0,Y 422.716,Z 736.909,A -85,B 0,C 180,E1 14277.685,E2 14277.685} C_VEL
LIN {X 0,Y 425.679,Z 718.457,A -85,B 0,C 180,E1 14275.848,E2 14275.848} C_VEL
LIN {X 0,Y 428.761,Z 698.397,A -85,B 0,C 180,E1 14274.173,E2 14274.173} C_VEL
LIN {X 0,Y 431.474,Z 679.137,A -85,B 0,C 180,E1 14272.833,E2 14272.833} C_VEL
LIN {X 0,Y 434.038,Z 658.178,A -85,B 0,C 180,E1 14271.664,E2 14271.664} C_VEL
LIN {X 0,Y 436.277,Z 636.719,A -85,B 0,C 180,E1 14270.726,E2 14270.726} C_VEL
LIN {X 0,Y 438.067,Z 615.512,A -85,B 0,C 180,E1 14270.033,E2 14270.033} C_VEL
LIN {X 0,Y 439.217,Z 593.245,A -85,B 0,C 180,E1 14269.534,E2 14269.534} C_VEL
LIN {X 0,Y 445.459,Z 373.069,A -85,B 0,C 180,E1 14265.64,E2 14265.64} C_VEL
LIN {X 0,Y 446.428,Z 336.454,A -85,B 0,C 180,E1 14264.955,E2 14264.955} C_VEL
LIN {X 0,Y 445.202,Z 327.777,A -85,B 0,C 180,E1 14264.615,E2 14264.615} C_VEL
LIN {X 0,Y 434.362,Z 309.52,A -85,B 0,C 180,E1 14262.816,E2 14262.816} C_VEL
LIN {X 0,Y 429.226,Z 301.233,A -85,B 0,C 180,E1 14261.866,E2 14261.866} C_VEL
LIN {X 0,Y 422.955,Z 287.999,A -85,B 0,C 180,E1 14259.488,E2 14259.488} C_VEL
LIN {X 0,Y 418.473,Z 279.237,A -85,B 0,C 180,E1 14257.71,E2 14257.71} C_VEL
LIN {X 0,Y 416.143,Z 274.848,A -85,B 0,C 180,E1 14256.747,E2 14256.747} C_VEL
LIN {X 0,Y 414.252,Z 271.107,A -85,B 0,C 180,E1 14255.911,E2 14255.911} C_VEL
LIN {X 0,Y 412.364,Z 267.62,A -85,B 0,C 180,E1 14255.076,E2 14255.076} C_VEL
LIN {X 0,Y 411.392,Z 266.061,A -85,B 0,C 180,E1 14254.662,E2 14254.662} C_VEL
LIN {X 0,Y 409.627,Z 262.72,A -85,B 0,C 180,E1 14253.817,E2 14253.817} C_VEL
LIN {X 0,Y 409.443,Z 261.755,A -85,B 0,C 180,E1 14253.414,E2 14253.414} C_VEL
LIN {X 0,Y 409.438,Z 261.727,A -85,B 0,C 180,E1 14249.558,E2 14249.558} C_VEL
LIN {X 0,Y 409.434,Z 261.729,A -85,B 0,C 180,E1 14245.611,E2 14245.611} C_VEL
LIN {X 0,Y 409.434,Z 261.733,A -85,B 0,C 180,E1 14241.639,E2 14241.639} C_VEL
LIN {X 0,Y 409.432,Z 261.724,A -85,B 0,C 180,E1 14237.746,E2 14237.746} C_VEL
LIN {X 0,Y 409.436,Z 261.724,A -85,B 0,C 180,E1 14233.847,E2 14233.847} C_VEL
LIN {X 0,Y 409.437,Z 261.728,A -85,B 0,C 180,E1 14229.986,E2 14229.986} C_VEL
LIN {X 0,Y 409.44,Z 261.736,A -85,B 0,C 180,E1 14226.029,E2 14226.029} C_VEL
LIN {X 0,Y 409.442,Z 261.726,A -85,B 0,C 180,E1 14222.1,E2 14222.1} C_VEL
LIN {X 0,Y 409.441,Z 261.724,A -85,B 0,C 180,E1 14218.182,E2 14218.182} C_VEL
LIN {X 0,Y 409.442,Z 261.735,A -85,B 0,C 180,E1 14214.255,E2 14214.255} C_VEL
LIN {X 0,Y 409.426,Z 261.728,A -85,B 0,C 180,E1 14210.442,E2 14210.442} C_VEL
LIN {X 0,Y 409.44,Z 261.884,A -85,B 0,C 180,E1 14207.735,E2 14207.735} C_VEL
LIN {X 0,Y 410.235,Z 264.436,A -85,B 0,C 180,E1 14207.044,E2 14207.044} C_VEL
LIN {X 0,Y 412.046,Z 267.091,A -85,B 0,C 180,E1 14206.244,E2 14206.244} C_VEL
LIN {X 0,Y 413.887,Z 270.838,A -85,B 0,C 180,E1 14205.307,E2 14205.307} C_VEL
LIN {X 0,Y 418.914,Z 280.932,A -85,B 0,C 180,E1 14202.929,E2 14202.929} C_VEL
LIN {X 0,Y 424.603,Z 293.418,A -85,B 0,C 180,E1 14200.323,E2 14200.323} C_VEL
LIN {X 0,Y 427.808,Z 300.636,A -85,B 0,C 180,E1 14198.996,E2 14198.996} C_VEL
LIN {X 0,Y 438.122,Z 317.156,A -85,B 0,C 180,E1 14197.138,E2 14197.138} C_VEL
LIN {X 0,Y 442.541,Z 325.171,A -85,B 0,C 180,E1 14196.367,E2 14196.367} C_VEL
LIN {X 0,Y 444.124,Z 336.515,A -85,B 0,C 180,E1 14195.904,E2 14195.904} C_VEL
LIN {X 0,Y 435.861,Z 568.389,A -85,B 0,C 180,E1 14191.588,E2 14191.588} C_VEL
LIN {X 0,Y 434.495,Z 589.195,A -85,B 0,C 180,E1 14190.963,E2 14190.963} C_VEL
LIN {X 0,Y 432.715,Z 609.086,A -85,B 0,C 180,E1 14190.13,E2 14190.13} C_VEL
LIN {X 0,Y 430.528,Z 628.832,A -85,B 0,C 180,E1 14189.05,E2 14189.05} C_VEL
LIN {X 0,Y 428.189,Z 646.697,A -85,B 0,C 180,E1 14187.834,E2 14187.834} C_VEL
LIN {X 0,Y 425.508,Z 664.861,A -85,B 0,C 180,E1 14186.322,E2 14186.322} C_VEL
LIN {X 0,Y 422.708,Z 682.022,A -85,B 0,C 180,E1 14184.586,E2 14184.586} C_VEL
LIN {X 0,Y 419.979,Z 697.798,A -85,B 0,C 180,E1 14182.672,E2 14182.672} C_VEL
LIN {X 0,Y 417.404,Z 712.201,A -85,B 0,C 180,E1 14180.598,E2 14180.598} C_VEL
LIN {X 0,Y 415.039,Z 725.545,A -85,B 0,C 180,E1 14178.316,E2 14178.316} C_VEL
LIN {X 0,Y 412.998,Z 737.507,A -85,B 0,C 180,E1 14175.88,E2 14175.88} C_VEL
LIN {X 0,Y 411.248,Z 748.496,A -85,B 0,C 180,E1 14173.168,E2 14173.168} C_VEL
LIN {X 0,Y 409.914,Z 757.961,A -85,B 0,C 180,E1 14170.271,E2 14170.271} C_VEL
LIN {X 0,Y 409.042,Z 765.309,A -85,B 0,C 180,E1 14167.402,E2 14167.402} C_VEL
LIN {X 0,Y 408.663,Z 769.356,A -85,B 0,C 180,E1 14165.419,E2 14165.419} C_VEL
LIN {X 0,Y 407.53,Z 771.271,A -85,B 0,C 180,E1 14164.372,E2 14164.372} C_VEL
LIN {X 0,Y 400.973,Z 775.779,A -85,B 0,C 180,E1 14161.49,E2 14161.49} C_VEL
LIN {X 0,Y 400.27,Z 776.591,A -85,B 0,C 180,E1 14160.626,E2 14160.626} C_VEL
LIN {X 0,Y 400.189,Z 778.276,A -85,B 0,C 180,E1 14157.693,E2 14157.693} C_VEL
LIN {X 0,Y 400.174,Z 778.336,A -85,B 0,C 180,E1 14154.821,E2 14154.821} C_VEL
LIN {X 0,Y 400.223,Z 776.853,A -85,B 0,C 180,E1 14151.855,E2 14151.855} C_VEL
LIN {X 0,Y 400.387,Z 773.84,A -85,B 0,C 180,E1 14148.945,E2 14148.945} C_VEL
LIN {X 0,Y 400.743,Z 769.315,A -85,B 0,C 180,E1 14146.079,E2 14146.079} C_VEL
LIN {X 0,Y 401.425,Z 762.791,A -85,B 0,C 180,E1 14143.102,E2 14143.102} C_VEL
LIN {X 0,Y 402.445,Z 754.871,A -85,B 0,C 180,E1 14140.306,E2 14140.306} C_VEL
LIN {X 0,Y 403.92,Z 745.158,A -85,B 0,C 180,E1 14137.54,E2 14137.54} C_VEL
LIN {X 0,Y 405.899,Z 733.412,A -85,B 0,C 180,E1 14134.806,E2 14134.806} C_VEL
LIN {X 0,Y 408.25,Z 720.269,A -85,B 0,C 180,E1 14132.28,E2 14132.28} C_VEL
LIN {X 0,Y 410.84,Z 706.077,A -85,B 0,C 180,E1 14130.001,E2 14130.001} C_VEL
LIN {X 0,Y 413.63,Z 690.635,A -85,B 0,C 180,E1 14127.924,E2 14127.924} C_VEL
LIN {X 0,Y 416.551,Z 673.564,A -85,B 0,C 180,E1 14126.01,E2 14126.01} C_VEL
LIN {X 0,Y 419.308,Z 656.079,A -85,B 0,C 180,E1 14124.391,E2 14124.391} C_VEL
LIN {X 0,Y 421.918,Z 637.736,A -85,B 0,C 180,E1 14122.991,E2 14122.991} C_VEL
LIN {X 0,Y 424.29,Z 618.498,A -85,B 0,C 180,E1 14121.805,E2 14121.805} C_VEL
LIN {X 0,Y 426.318,Z 598.645,A -85,B 0,C 180,E1 14120.846,E2 14120.846} C_VEL
LIN {X 0,Y 427.933,Z 578.046,A -85,B 0,C 180,E1 14120.105,E2 14120.105} C_VEL
LIN {X 0,Y 429.051,Z 556.092,A -85,B 0,C 180,E1 14119.58,E2 14119.58} C_VEL
LIN {X 0,Y 436.287,Z 336.164,A -85,B 0,C 180,E1 14115.557,E2 14115.557} C_VEL
LIN {X 0,Y 434.493,Z 326.317,A -85,B 0,C 180,E1 14115.122,E2 14115.122} C_VEL
LIN {X 0,Y 421.95,Z 305.298,A -85,B 0,C 180,E1 14113.036,E2 14113.036} C_VEL
LIN {X 0,Y 418.204,Z 299.217,A -85,B 0,C 180,E1 14112.326,E2 14112.326} C_VEL
LIN {X 0,Y 411.33,Z 283.52,A -85,B 0,C 180,E1 14109.361,E2 14109.361} C_VEL
LIN {X 0,Y 405.416,Z 271.146,A -85,B 0,C 180,E1 14106.761,E2 14106.761} C_VEL
LIN {X 0,Y 402.938,Z 266.353,A -85,B 0,C 180,E1 14105.677,E2 14105.677} C_VEL
LIN {X 0,Y 401.527,Z 262.964,A -85,B 0,C 180,E1 14104.879,E2 14104.879} C_VEL
LIN {X 0,Y 401.503,Z 262.708,A -85,B 0,C 180,E1 14101.763,E2 14101.763} C_VEL
LIN {X 0,Y 401.499,Z 262.707,A -85,B 0,C 180,E1 14097.799,E2 14097.799} C_VEL
LIN {X 0,Y 401.5,Z 262.706,A -85,B 0,C 180,E1 14093.787,E2 14093.787} C_VEL
LIN {X 0,Y 401.503,Z 262.703,A -85,B 0,C 180,E1 14089.838,E2 14089.838} C_VEL
LIN {X 0,Y 401.501,Z 262.702,A -85,B 0,C 180,E1 14085.822,E2 14085.822} C_VEL
LIN {X 0,Y 401.5,Z 262.705,A -85,B 0,C 180,E1 14081.864,E2 14081.864} C_VEL
LIN {X 0,Y 401.504,Z 262.719,A -85,B 0,C 180,E1 14077.872,E2 14077.872} C_VEL
LIN {X 0,Y 401.503,Z 262.718,A -85,B 0,C 180,E1 14073.903,E2 14073.903} C_VEL
LIN {X 0,Y 401.508,Z 262.701,A -85,B 0,C 180,E1 14069.869,E2 14069.869} C_VEL
LIN {X 0,Y 401.496,Z 262.703,A -85,B 0,C 180,E1 14065.976,E2 14065.976} C_VEL
LIN {X 0,Y 401.492,Z 262.722,A -85,B 0,C 180,E1 14062.087,E2 14062.087} C_VEL
LIN {X 0,Y 401.486,Z 262.712,A -85,B 0,C 180,E1 14058.136,E2 14058.136} C_VEL
LIN {X 0,Y 401.477,Z 262.695,A -85,B 0,C 180,E1 14054.272,E2 14054.272} C_VEL
LIN {X 0,Y 401.48,Z 262.719,A -85,B 0,C 180,E1 14050.328,E2 14050.328} C_VEL
LIN {X 0,Y 401.48,Z 262.724,A -85,B 0,C 180,E1 14046.29,E2 14046.29} C_VEL
LIN {X 0,Y 401.477,Z 262.703,A -85,B 0,C 180,E1 14042.282,E2 14042.282} C_VEL
LIN {X 0,Y 401.482,Z 262.705,A -85,B 0,C 180,E1 14038.429,E2 14038.429} C_VEL
LIN {X 0,Y 401.485,Z 262.72,A -85,B 0,C 180,E1 14034.425,E2 14034.425} C_VEL
LIN {X 0,Y 401.491,Z 262.719,A -85,B 0,C 180,E1 14030.539,E2 14030.539} C_VEL
LIN {X 0,Y 401.499,Z 262.705,A -85,B 0,C 180,E1 14026.608,E2 14026.608} C_VEL
LIN {X 0,Y 401.501,Z 262.703,A -85,B 0,C 180,E1 14022.761,E2 14022.761} C_VEL
LIN {X 0,Y 401.505,Z 262.703,A -85,B 0,C 180,E1 14018.832,E2 14018.832} C_VEL
LIN {X 0,Y 401.501,Z 262.705,A -85,B 0,C 180,E1 14014.953,E2 14014.953} C_VEL
LIN {X 0,Y 401.504,Z 262.706,A -85,B 0,C 180,E1 14010.947,E2 14010.947} C_VEL
LIN {X 0,Y 401.501,Z 262.742,A -85,B 0,C 180,E1 14006.949,E2 14006.949} C_VEL
LIN {X 0,Y 401.652,Z 263.547,A -85,B 0,C 180,E1 14006.579,E2 14006.579} C_VEL
LIN {X 0,Y 403.142,Z 266.691,A -85,B 0,C 180,E1 14005.908,E2 14005.908} C_VEL
LIN {X 0,Y 404.349,Z 268.824,A -85,B 0,C 180,E1 14005.426,E2 14005.426} C_VEL
LIN {X 0,Y 406.758,Z 273.403,A -85,B 0,C 180,E1 14004.449,E2 14004.449} C_VEL
LIN {X 0,Y 413.359,Z 286.105,A -85,B 0,C 180,E1 14001.916,E2 14001.916} C_VEL
LIN {X 0,Y 421.143,Z 301.99,A -85,B 0,C 180,E1 13999.104,E2 13999.104} C_VEL
LIN {X 0,Y 433.641,Z 321.771,A -85,B 0,C 180,E1 13996.983,E2 13996.983} C_VEL
LIN {X 0,Y 440.074,Z 332.946,A -85,B 0,C 180,E1 13995.941,E2 13995.941} C_VEL
LIN {X 0,Y 440.821,Z 340.498,A -85,B 0,C 180,E1 13995.685,E2 13995.685} C_VEL
LIN {X 0,Y 434.343,Z 552.887,A -85,B 0,C 180,E1 13991.884,E2 13991.884} C_VEL
LIN {X 0,Y 432.672,Z 605.426,A -85,B 0,C 180,E1 13990.919,E2 13990.919} C_VEL
LIN {X 0,Y 430.989,Z 627.599,A -85,B 0,C 180,E1 13990.3,E2 13990.3} C_VEL
LIN {X 0,Y 428.915,Z 648.601,A -85,B 0,C 180,E1 13989.478,E2 13989.478} C_VEL
LIN {X 0,Y 426.415,Z 669.619,A -85,B 0,C 180,E1 13988.414,E2 13988.414} C_VEL
LIN {X 0,Y 423.644,Z 689.272,A -85,B 0,C 180,E1 13987.169,E2 13987.169} C_VEL
LIN {X 0,Y 420.657,Z 708.325,A -85,B 0,C 180,E1 13985.697,E2 13985.697} C_VEL
LIN {X 0,Y 417.588,Z 726.873,A -85,B 0,C 180,E1 13983.99,E2 13983.99} C_VEL
LIN {X 0,Y 414.439,Z 744.589,A -85,B 0,C 180,E1 13982.055,E2 13982.055} C_VEL
LIN {X 0,Y 411.418,Z 761.409,A -85,B 0,C 180,E1 13979.879,E2 13979.879} C_VEL
LIN {X 0,Y 408.502,Z 777.772,A -85,B 0,C 180,E1 13977.395,E2 13977.395} C_VEL
LIN {X 0,Y 406.117,Z 791.843,A -85,B 0,C 180,E1 13974.896,E2 13974.896} C_VEL
LIN {X 0,Y 404.111,Z 804.449,A -85,B 0,C 180,E1 13972.242,E2 13972.242} C_VEL
LIN {X 0,Y 402.46,Z 816.311,A -85,B 0,C 180,E1 13969.293,E2 13969.293} C_VEL
LIN {X 0,Y 401.321,Z 826.185,A -85,B 0,C 180,E1 13966.35,E2 13966.35} C_VEL
LIN {X 0,Y 400.602,Z 834.169,A -85,B 0,C 180,E1 13963.42,E2 13963.42} C_VEL
LIN {X 0,Y 400.204,Z 840.717,A -85,B 0,C 180,E1 13960.361,E2 13960.361} C_VEL
LIN {X 0,Y 400.032,Z 845.406,A -85,B 0,C 180,E1 13957.466,E2 13957.466} C_VEL
LIN {X 0,Y 399.996,Z 848.435,A -85,B 0,C 180,E1 13954.586,E2 13954.586} C_VEL
LIN {X 0,Y 399.991,Z 850.113,A -85,B 0,C 180,E1 13951.574,E2 13951.574} C_VEL
LIN {X 0,Y 400.001,Z 850.174,A -85,B 0,C 180,E1 13948.853,E2 13948.853} C_VEL
LIN {X 0,Y 399.996,Z 848.745,A -85,B 0,C 180,E1 13945.841,E2 13945.841} C_VEL
LIN {X 0,Y 400.033,Z 846.005,A -85,B 0,C 180,E1 13943.108,E2 13943.108} C_VEL
LIN {X 0,Y 400.168,Z 841.391,A -85,B 0,C 180,E1 13940.071,E2 13940.071} C_VEL
LIN {X 0,Y 400.506,Z 835.398,A -85,B 0,C 180,E1 13937.161,E2 13937.161} C_VEL
LIN {X 0,Y 401.168,Z 827.43,A -85,B 0,C 180,E1 13934.167,E2 13934.167} C_VEL
LIN {X 0,Y 402.245,Z 817.567,A -85,B 0,C 180,E1 13931.146,E2 13931.146} C_VEL
LIN {X 0,Y 403.719,Z 806.591,A -85,B 0,C 180,E1 13928.344,E2 13928.344} C_VEL
LIN {X 0,Y 405.585,Z 794.175,A -85,B 0,C 180,E1 13925.687,E2 13925.687} C_VEL
LIN {X 0,Y 407.976,Z 779.672,A -85,B 0,C 180,E1 13923.037,E2 13923.037} C_VEL
LIN {X 0,Y 410.623,Z 764.476,A -85,B 0,C 180,E1 13920.66,E2 13920.66} C_VEL
LIN {X 0,Y 413.602,Z 747.618,A -85,B 0,C 180,E1 13918.428,E2 13918.428} C_VEL
LIN {X 0,Y 416.71,Z 729.794,A -85,B 0,C 180,E1 13916.421,E2 13916.421} C_VEL
LIN {X 0,Y 419.853,Z 711.127,A -85,B 0,C 180,E1 13914.64,E2 13914.64} C_VEL
LIN {X 0,Y 422.91,Z 691.695,A -85,B 0,C 180,E1 13913.092,E2 13913.092} C_VEL
LIN {X 0,Y 425.72,Z 671.828,A -85,B 0,C 180,E1 13911.797,E2 13911.797} C_VEL
LIN {X 0,Y 428.372,Z 650.451,A -85,B 0,C 180,E1 13910.675,E2 13910.675} C_VEL
LIN {X 0,Y 430.541,Z 629.355,A -85,B 0,C 180,E1 13909.816,E2 13909.816} C_VEL
LIN {X 0,Y 432.23,Z 607.309,A -85,B 0,C 180,E1 13909.181,E2 13909.181} C_VEL
LIN {X 0,Y 433.407,Z 576.201,A -85,B 0,C 180,E1 13908.576,E2 13908.576} C_VEL
LIN {X 0,Y 439.871,Z 363.621,A -85,B 0,C 180,E1 13904.765,E2 13904.765} C_VEL
LIN {X 0,Y 440.549,Z 337.886,A -85,B 0,C 180,E1 13904.27,E2 13904.27} C_VEL
LIN {X 0,Y 439.617,Z 331.695,A -85,B 0,C 180,E1 13904.014,E2 13904.014} C_VEL
LIN {X 0,Y 428.91,Z 313.403,A -85,B 0,C 180,E1 13902.156,E2 13902.156} C_VEL
LIN {X 0,Y 421.106,Z 301.202,A -85,B 0,C 180,E1 13900.675,E2 13900.675} C_VEL
LIN {X 0,Y 415.404,Z 289.306,A -85,B 0,C 180,E1 13898.389,E2 13898.389} C_VEL
LIN {X 0,Y 411.094,Z 280.937,A -85,B 0,C 180,E1 13896.577,E2 13896.577} C_VEL
LIN {X 0,Y 408.517,Z 276.208,A -85,B 0,C 180,E1 13895.456,E2 13895.456} C_VEL
LIN {X 0,Y 406.397,Z 272.165,A -85,B 0,C 180,E1 13894.463,E2 13894.463} C_VEL
LIN {X 0,Y 404.6,Z 268.92,A -85,B 0,C 180,E1 13893.611,E2 13893.611} C_VEL
LIN {X 0,Y 403.727,Z 267.334,A -85,B 0,C 180,E1 13893.184,E2 13893.184} C_VEL
LIN {X 0,Y 401.932,Z 264.516,A -85,B 0,C 180,E1 13892.334,E2 13892.334} C_VEL
LIN {X 0,Y 401.518,Z 262.827,A -85,B 0,C 180,E1 13891.82,E2 13891.82} C_VEL
LIN {X 0,Y 401.505,Z 262.723,A -85,B 0,C 180,E1 13887.863,E2 13887.863} C_VEL
LIN {X 0,Y 401.5,Z 262.714,A -85,B 0,C 180,E1 13883.942,E2 13883.942} C_VEL
LIN {X 0,Y 401.5,Z 262.713,A -85,B 0,C 180,E1 13880.101,E2 13880.101} C_VEL
LIN {X 0,Y 401.502,Z 262.72,A -85,B 0,C 180,E1 13876.196,E2 13876.196} C_VEL
LIN {X 0,Y 401.502,Z 262.72,A -85,B 0,C 180,E1 13872.222,E2 13872.222} C_VEL
LIN {X 0,Y 401.506,Z 262.711,A -85,B 0,C 180,E1 13868.161,E2 13868.161} C_VEL
LIN {X 0,Y 401.5,Z 262.712,A -85,B 0,C 180,E1 13864.143,E2 13864.143} C_VEL
LIN {X 0,Y 401.51,Z 262.721,A -85,B 0,C 180,E1 13860.144,E2 13860.144} C_VEL
LIN {X 0,Y 401.499,Z 262.716,A -85,B 0,C 180,E1 13856.146,E2 13856.146} C_VEL
LIN {X 0,Y 401.507,Z 262.716,A -85,B 0,C 180,E1 13852.129,E2 13852.129} C_VEL
LIN {X 0,Y 401.496,Z 262.953,A -85,B 0,C 180,E1 13849.382,E2 13849.382} C_VEL
LIN {X 0,Y 402.84,Z 266.272,A -85,B 0,C 180,E1 13848.403,E2 13848.403} C_VEL
LIN {X 0,Y 404.263,Z 268.426,A -85,B 0,C 180,E1 13847.721,E2 13847.721} C_VEL
LIN {X 0,Y 406.056,Z 271.904,A -85,B 0,C 180,E1 13846.763,E2 13846.763} C_VEL
LIN {X 0,Y 409.496,Z 278.723,A -85,B 0,C 180,E1 13845.001,E2 13845.001} C_VEL
LIN {X 0,Y 414.813,Z 289.52,A -85,B 0,C 180,E1 13842.466,E2 13842.466} C_VEL
LIN {X 0,Y 419.855,Z 300.644,A -85,B 0,C 180,E1 13840.2,E2 13840.2} C_VEL
LIN {X 0,Y 430.753,Z 317.935,A -85,B 0,C 180,E1 13838.129,E2 13838.129} C_VEL
LIN {X 0,Y 437.2,Z 329.334,A -85,B 0,C 180,E1 13836.963,E2 13836.963} C_VEL
LIN {X 0,Y 438.328,Z 338.071,A -85,B 0,C 180,E1 13836.603,E2 13836.603} C_VEL
LIN {X 0,Y 429.621,Z 568.918,A -85,B 0,C 180,E1 13832.247,E2 13832.247} C_VEL
LIN {X 0,Y 428.187,Z 589.731,A -85,B 0,C 180,E1 13831.614,E2 13831.614} C_VEL
LIN {X 0,Y 426.286,Z 609.917,A -85,B 0,C 180,E1 13830.756,E2 13830.756} C_VEL
LIN {X 0,Y 423.998,Z 629.544,A -85,B 0,C 180,E1 13829.667,E2 13829.667} C_VEL
LIN {X 0,Y 421.432,Z 648.121,A -85,B 0,C 180,E1 13828.379,E2 13828.379} C_VEL
LIN {X 0,Y 418.776,Z 665.23,A -85,B 0,C 180,E1 13826.935,E2 13826.935} C_VEL
LIN {X 0,Y 415.873,Z 682.128,A -85,B 0,C 180,E1 13825.206,E2 13825.206} C_VEL
LIN {X 0,Y 412.969,Z 697.991,A -85,B 0,C 180,E1 13823.265,E2 13823.265} C_VEL
LIN {X 0,Y 410.11,Z 713.135,A -85,B 0,C 180,E1 13821.055,E2 13821.055} C_VEL
LIN {X 0,Y 407.526,Z 726.837,A -85,B 0,C 180,E1 13818.658,E2 13818.658} C_VEL
LIN {X 0,Y 405.438,Z 738.306,A -85,B 0,C 180,E1 13816.269,E2 13816.269} C_VEL
LIN {X 0,Y 403.578,Z 749.193,A -85,B 0,C 180,E1 13813.532,E2 13813.532} C_VEL
LIN {X 0,Y 402.157,Z 758.456,A -85,B 0,C 180,E1 13810.648,E2 13810.648} C_VEL
LIN {X 0,Y 401.219,Z 765.648,A -85,B 0,C 180,E1 13807.811,E2 13807.811} C_VEL
LIN {X 0,Y 400.657,Z 771.063,A -85,B 0,C 180,E1 13805.029,E2 13805.029} C_VEL
LIN {X 0,Y 400.353,Z 775.102,A -85,B 0,C 180,E1 13802.139,E2 13802.139} C_VEL
LIN {X 0,Y 400.27,Z 776.591,A -85,B 0,C 180,E1 13800.626,E2 13800.626} C_VEL
LIN {X 0,Y 399.213,Z 777.51,A -85,B 0,C 180,E1 13799.53,E2 13799.53} C_VEL
LIN {X 0,Y 392.843,Z 779.183,A -85,B 0,C 180,E1 13796.515,E2 13796.515} C_VEL
LIN {X 0,Y 392.204,Z 779.192,A -85,B 0,C 180,E1 13795.624,E2 13795.624} C_VEL
LIN {X 0,Y 392.244,Z 778.204,A -85,B 0,C 180,E1 13792.64,E2 13792.64} C_VEL
LIN {X 0,Y 392.377,Z 775.578,A -85,B 0,C 180,E1 13789.657,E2 13789.657} C_VEL
LIN {X 0,Y 392.694,Z 771.439,A -85,B 0,C 180,E1 13786.723,E2 13786.723} C_VEL
LIN {X 0,Y 393.329,Z 765.421,A -85,B 0,C 180,E1 13783.676,E2 13783.676} C_VEL
LIN {X 0,Y 394.321,Z 758.049,A -85,B 0,C 180,E1 13780.816,E2 13780.816} C_VEL
LIN {X 0,Y 395.767,Z 748.908,A -85,B 0,C 180,E1 13777.985,E2 13777.985} C_VEL
LIN {X 0,Y 397.716,Z 737.786,A -85,B 0,C 180,E1 13775.194,E2 13775.194} C_VEL
LIN {X 0,Y 399.934,Z 725.871,A -85,B 0,C 180,E1 13772.724,E2 13772.724} C_VEL
LIN {X 0,Y 402.45,Z 712.718,A -85,B 0,C 180,E1 13770.429,E2 13770.429} C_VEL
LIN {X 0,Y 405.311,Z 697.773,A -85,B 0,C 180,E1 13768.234,E2 13768.234} C_VEL
LIN {X 0,Y 408.258,Z 681.907,A -85,B 0,C 180,E1 13766.28,E2 13766.28} C_VEL
LIN {X 0,Y 411.275,Z 664.472,A -85,B 0,C 180,E1 13764.491,E2 13764.491} C_VEL
LIN {X 0,Y 414.193,Z 645.887,A -85,B 0,C 180,E1 13762.93,E2 13762.93} C_VEL
LIN {X 0,Y 416.754,Z 627.216,A -85,B 0,C 180,E1 13761.656,E2 13761.656} C_VEL
LIN {X 0,Y 419.062,Z 607.023,A -85,B 0,C 180,E1 13760.56,E2 13760.56} C_VEL
LIN {X 0,Y 421.012,Z 585.812,A -85,B 0,C 180,E1 13759.698,E2 13759.698} C_VEL
LIN {X 0,Y 422.332,Z 565.342,A -85,B 0,C 180,E1 13759.11,E2 13759.11} C_VEL
LIN {X 0,Y 430.355,Z 337.945,A -85,B 0,C 180,E1 13754.88,E2 13754.88} C_VEL
LIN {X 0,Y 428.96,Z 330.401,A -85,B 0,C 180,E1 13754.534,E2 13754.534} C_VEL
LIN {X 0,Y 417.096,Z 310.411,A -85,B 0,C 180,E1 13752.5,E2 13752.5} C_VEL
LIN {X 0,Y 410.22,Z 299.514,A -85,B 0,C 180,E1 13751.234,E2 13751.234} C_VEL
LIN {X 0,Y 403.565,Z 284.684,A -85,B 0,C 180,E1 13748.287,E2 13748.287} C_VEL
LIN {X 0,Y 397.575,Z 272.227,A -85,B 0,C 180,E1 13745.554,E2 13745.554} C_VEL
LIN {X 0,Y 395.128,Z 267.529,A -85,B 0,C 180,E1 13744.432,E2 13744.432} C_VEL
LIN {X 0,Y 393.582,Z 263.901,A -85,B 0,C 180,E1 13743.525,E2 13743.525} C_VEL
LIN {X 0,Y 393.567,Z 263.712,A -85,B 0,C 180,E1 13739.634,E2 13739.634} C_VEL
LIN {X 0,Y 393.561,Z 263.706,A -85,B 0,C 180,E1 13735.654,E2 13735.654} C_VEL
LIN {X 0,Y 393.566,Z 263.706,A -85,B 0,C 180,E1 13731.695,E2 13731.695} C_VEL
LIN {X 0,Y 393.563,Z 263.711,A -85,B 0,C 180,E1 13727.669,E2 13727.669} C_VEL
LIN {X 0,Y 393.563,Z 263.711,A -85,B 0,C 180,E1 13723.613,E2 13723.613} C_VEL
LIN {X 0,Y 393.565,Z 263.699,A -85,B 0,C 180,E1 13719.616,E2 13719.616} C_VEL
LIN {X 0,Y 393.559,Z 263.686,A -85,B 0,C 180,E1 13715.574,E2 13715.574} C_VEL
LIN {X 0,Y 393.565,Z 263.689,A -85,B 0,C 180,E1 13711.555,E2 13711.555} C_VEL
LIN {X 0,Y 393.567,Z 263.712,A -85,B 0,C 180,E1 13707.538,E2 13707.538} C_VEL
LIN {X 0,Y 393.566,Z 263.702,A -85,B 0,C 180,E1 13703.496,E2 13703.496} C_VEL
LIN {X 0,Y 393.561,Z 263.683,A -85,B 0,C 180,E1 13699.524,E2 13699.524} C_VEL
LIN {X 0,Y 393.566,Z 263.696,A -85,B 0,C 180,E1 13695.47,E2 13695.47} C_VEL
LIN {X 0,Y 393.563,Z 263.709,A -85,B 0,C 180,E1 13691.428,E2 13691.428} C_VEL
LIN {X 0,Y 393.565,Z 263.69,A -85,B 0,C 180,E1 13687.443,E2 13687.443} C_VEL
LIN {X 0,Y 393.557,Z 263.69,A -85,B 0,C 180,E1 13683.494,E2 13683.494} C_VEL
LIN {X 0,Y 393.569,Z 263.707,A -85,B 0,C 180,E1 13679.417,E2 13679.417} C_VEL
LIN {X 0,Y 393.56,Z 263.708,A -85,B 0,C 180,E1 13675.336,E2 13675.336} C_VEL
LIN {X 0,Y 393.558,Z 263.695,A -85,B 0,C 180,E1 13671.378,E2 13671.378} C_VEL
LIN {X 0,Y 393.553,Z 263.687,A -85,B 0,C 180,E1 13667.379,E2 13667.379} C_VEL
LIN {X 0,Y 393.547,Z 263.693,A -85,B 0,C 180,E1 13663.467,E2 13663.467} C_VEL
LIN {X 0,Y 393.544,Z 263.698,A -85,B 0,C 180,E1 13659.474,E2 13659.474} C_VEL
LIN {X 0,Y 393.54,Z 263.699,A -85,B 0,C 180,E1 13655.535,E2 13655.535} C_VEL
LIN {X 0,Y 393.541,Z 263.697,A -85,B 0,C 180,E1 13651.526,E2 13651.526} C_VEL
LIN {X 0,Y 393.581,Z 263.907,A -85,B 0,C 180,E1 13648.156,E2 13648.156} C_VEL
LIN {X 0,Y 394.882,Z 267.238,A -85,B 0,C 180,E1 13647.361,E2 13647.361} C_VEL
LIN {X 0,Y 396.311,Z 269.447,A -85,B 0,C 180,E1 13646.805,E2 13646.805} C_VEL
LIN {X 0,Y 401.681,Z 279.798,A -85,B 0,C 180,E1 13644.55,E2 13644.55} C_VEL
LIN {X 0,Y 407.911,Z 291.861,A -85,B 0,C 180,E1 13642.115,E2 13642.115} C_VEL
LIN {X 0,Y 413.093,Z 302.276,A -85,B 0,C 180,E1 13640.238,E2 13640.238} C_VEL
LIN {X 0,Y 426.197,Z 322.63,A -85,B 0,C 180,E1 13637.926,E2 13637.926} C_VEL
LIN {X 0,Y 434.475,Z 336.841,A -85,B 0,C 180,E1 13636.537,E2 13636.537} C_VEL
LIN {X 0,Y 434.886,Z 342.077,A -85,B 0,C 180,E1 13636.369,E2 13636.369} C_VEL
LIN {X 0,Y 428.057,Z 554.712,A -85,B 0,C 180,E1 13632.521,E2 13632.521} C_VEL
LIN {X 0,Y 426.369,Z 605.161,A -85,B 0,C 180,E1 13631.582,E2 13631.582} C_VEL
LIN {X 0,Y 424.625,Z 627.25,A -85,B 0,C 180,E1 13630.961,E2 13630.961} C_VEL
LIN {X 0,Y 422.486,Z 647.997,A -85,B 0,C 180,E1 13630.144,E2 13630.144} C_VEL
LIN {X 0,Y 419.904,Z 668.877,A -85,B 0,C 180,E1 13629.08,E2 13629.08} C_VEL
LIN {X 0,Y 417.077,Z 688.057,A -85,B 0,C 180,E1 13627.856,E2 13627.856} C_VEL
LIN {X 0,Y 413.788,Z 708.07,A -85,B 0,C 180,E1 13626.297,E2 13626.297} C_VEL
LIN {X 0,Y 410.435,Z 727.25,A -85,B 0,C 180,E1 13624.497,E2 13624.497} C_VEL
LIN {X 0,Y 407.076,Z 745.329,A -85,B 0,C 180,E1 13622.482,E2 13622.482} C_VEL
LIN {X 0,Y 403.983,Z 761.591,A -85,B 0,C 180,E1 13620.323,E2 13620.323} C_VEL
LIN {X 0,Y 400.918,Z 777.821,A -85,B 0,C 180,E1 13617.796,E2 13617.796} C_VEL
LIN {X 0,Y 398.411,Z 791.775,A -85,B 0,C 180,E1 13615.252,E2 13615.252} C_VEL
LIN {X 0,Y 396.204,Z 804.99,A -85,B 0,C 180,E1 13612.398,E2 13612.398} C_VEL
LIN {X 0,Y 394.542,Z 816.295,A -85,B 0,C 180,E1 13609.484,E2 13609.484} C_VEL
LIN {X 0,Y 393.325,Z 826.298,A -85,B 0,C 180,E1 13606.388,E2 13606.388} C_VEL
LIN {X 0,Y 392.591,Z 834.244,A -85,B 0,C 180,E1 13603.372,E2 13603.372} C_VEL
LIN {X 0,Y 392.218,Z 840.265,A -85,B 0,C 180,E1 13600.426,E2 13600.426} C_VEL
LIN {X 0,Y 392.051,Z 845.036,A -85,B 0,C 180,E1 13597.324,E2 13597.324} C_VEL
LIN {X 0,Y 392.021,Z 847.845,A -85,B 0,C 180,E1 13594.533,E2 13594.533} C_VEL
LIN {X 0,Y 392.024,Z 849.426,A -85,B 0,C 180,E1 13591.46,E2 13591.46} C_VEL
LIN {X 0,Y 392.032,Z 849.455,A -85,B 0,C 180,E1 13588.804,E2 13588.804} C_VEL
LIN {X 0,Y 392.023,Z 848.016,A -85,B 0,C 180,E1 13585.753,E2 13585.753} C_VEL
LIN {X 0,Y 392.06,Z 845.268,A -85,B 0,C 180,E1 13582.967,E2 13582.967} C_VEL
LIN {X 0,Y 392.206,Z 840.425,A -85,B 0,C 180,E1 13579.75,E2 13579.75} C_VEL
LIN {X 0,Y 392.574,Z 834.3,A -85,B 0,C 180,E1 13576.747,E2 13576.747} C_VEL
LIN {X 0,Y 393.278,Z 826.402,A -85,B 0,C 180,E1 13573.759,E2 13573.759} C_VEL
LIN {X 0,Y 394.48,Z 816.202,A -85,B 0,C 180,E1 13570.606,E2 13570.606} C_VEL
LIN {X 0,Y 396.072,Z 805.11,A -85,B 0,C 180,E1 13567.748,E2 13567.748} C_VEL
LIN {X 0,Y 398.096,Z 792.569,A -85,B 0,C 180,E1 13565.041,E2 13565.041} C_VEL
LIN {X 0,Y 400.68,Z 777.885,A -85,B 0,C 180,E1 13562.344,E2 13562.344} C_VEL
LIN {X 0,Y 403.599,Z 762.151,A -85,B 0,C 180,E1 13559.88,E2 13559.88} C_VEL
LIN {X 0,Y 406.805,Z 745.02,A -85,B 0,C 180,E1 13557.6,E2 13557.6} C_VEL
LIN {X 0,Y 410.067,Z 727.271,A -85,B 0,C 180,E1 13555.617,E2 13555.617} C_VEL
LIN {X 0,Y 413.367,Z 708.399,A -85,B 0,C 180,E1 13553.828,E2 13553.828} C_VEL
LIN {X 0,Y 416.633,Z 688.638,A -85,B 0,C 180,E1 13552.267,E2 13552.267} C_VEL
LIN {X 0,Y 419.512,Z 669.033,A -85,B 0,C 180,E1 13551.007,E2 13551.007} C_VEL
LIN {X 0,Y 422.21,Z 647.532,A -85,B 0,C 180,E1 13549.898,E2 13549.898} C_VEL
LIN {X 0,Y 424.468,Z 625.936,A -85,B 0,C 180,E1 13549.046,E2 13549.046} C_VEL
LIN {X 0,Y 426.228,Z 603.675,A -85,B 0,C 180,E1 13548.423,E2 13548.423} C_VEL
LIN {X 0,Y 428.317,Z 539.503,A -85,B 0,C 180,E1 13547.24,E2 13547.24} C_VEL
LIN {X 0,Y 434.878,Z 340.366,A -85,B 0,C 180,E1 13543.606,E2 13543.606} C_VEL
LIN {X 0,Y 434.091,Z 335.536,A -85,B 0,C 180,E1 13543.391,E2 13543.391} C_VEL
LIN {X 0,Y 423.548,Z 317.517,A -85,B 0,C 180,E1 13541.489,E2 13541.489} C_VEL
LIN {X 0,Y 413.749,Z 302.427,A -85,B 0,C 180,E1 13539.574,E2 13539.574} C_VEL
LIN {X 0,Y 411.256,Z 297.577,A -85,B 0,C 180,E1 13538.67,E2 13538.67} C_VEL
LIN {X 0,Y 406.044,Z 287.024,A -85,B 0,C 180,E1 13536.403,E2 13536.403} C_VEL
LIN {X 0,Y 401.409,Z 278.264,A -85,B 0,C 180,E1 13534.26,E2 13534.26} C_VEL
LIN {X 0,Y 398.772,Z 273.475,A -85,B 0,C 180,E1 13532.964,E2 13532.964} C_VEL
LIN {X 0,Y 396.798,Z 270.042,A -85,B 0,C 180,E1 13531.95,E2 13531.95} C_VEL
LIN {X 0,Y 396.011,Z 268.536,A -85,B 0,C 180,E1 13531.51,E2 13531.51} C_VEL
LIN {X 0,Y 394.012,Z 265.552,A -85,B 0,C 180,E1 13530.5,E2 13530.5} C_VEL
LIN {X 0,Y 393.577,Z 263.783,A -85,B 0,C 180,E1 13529.877,E2 13529.877} C_VEL
LIN {X 0,Y 393.56,Z 263.703,A -85,B 0,C 180,E1 13525.912,E2 13525.912} C_VEL
LIN {X 0,Y 393.567,Z 263.712,A -85,B 0,C 180,E1 13521.93,E2 13521.93} C_VEL
LIN {X 0,Y 393.558,Z 263.701,A -85,B 0,C 180,E1 13517.904,E2 13517.904} C_VEL
LIN {X 0,Y 393.563,Z 263.699,A -85,B 0,C 180,E1 13513.952,E2 13513.952} C_VEL
LIN {X 0,Y 393.558,Z 263.706,A -85,B 0,C 180,E1 13509.949,E2 13509.949} C_VEL
LIN {X 0,Y 393.561,Z 263.712,A -85,B 0,C 180,E1 13505.98,E2 13505.98} C_VEL
LIN {X 0,Y 393.554,Z 263.702,A -85,B 0,C 180,E1 13501.894,E2 13501.894} C_VEL
LIN {X 0,Y 393.556,Z 263.702,A -85,B 0,C 180,E1 13497.963,E2 13497.963} C_VEL
LIN {X 0,Y 393.563,Z 263.713,A -85,B 0,C 180,E1 13494.022,E2 13494.022} C_VEL
LIN {X 0,Y 393.556,Z 263.926,A -85,B 0,C 180,E1 13491.307,E2 13491.307} C_VEL
LIN {X 0,Y 395.142,Z 267.574,A -85,B 0,C 180,E1 13490.093,E2 13490.093} C_VEL
LIN {X 0,Y 396.471,Z 269.558,A -85,B 0,C 180,E1 13489.393,E2 13489.393} C_VEL
LIN {X 0,Y 398.436,Z 273.195,A -85,B 0,C 180,E1 13488.273,E2 13488.273} C_VEL
LIN {X 0,Y 401.708,Z 279.653,A -85,B 0,C 180,E1 13486.471,E2 13486.471} C_VEL
LIN {X 0,Y 405.721,Z 287.634,A -85,B 0,C 180,E1 13484.419,E2 13484.419} C_VEL
LIN {X 0,Y 411.504,Z 300.186,A -85,B 0,C 180,E1 13481.588,E2 13481.588} C_VEL
LIN {X 0,Y 421.044,Z 314.927,A -85,B 0,C 180,E1 13479.625,E2 13479.625} C_VEL
LIN {X 0,Y 431.615,Z 332.612,A -85,B 0,C 180,E1 13477.637,E2 13477.637} C_VEL
LIN {X 0,Y 432.627,Z 339.558,A -85,B 0,C 180,E1 13477.325,E2 13477.325} C_VEL
LIN {X 0,Y 423.447,Z 569.425,A -85,B 0,C 180,E1 13472.927,E2 13472.927} C_VEL
LIN {X 0,Y 421.95,Z 590.225,A -85,B 0,C 180,E1 13472.287,E2 13472.287} C_VEL
LIN {X 0,Y 420.027,Z 609.79,A -85,B 0,C 180,E1 13471.451,E2 13471.451} C_VEL
LIN {X 0,Y 417.633,Z 629.537,A -85,B 0,C 180,E1 13470.351,E2 13470.351} C_VEL
LIN {X 0,Y 414.978,Z 647.975,A -85,B 0,C 180,E1 13469.067,E2 13469.067} C_VEL
LIN {X 0,Y 411.99,Z 666.21,A -85,B 0,C 180,E1 13467.51,E2 13467.51} C_VEL
LIN {X 0,Y 408.917,Z 683.237,A -85,B 0,C 180,E1 13465.738,E2 13465.738} C_VEL
LIN {X 0,Y 405.836,Z 699.146,A -85,B 0,C 180,E1 13463.754,E2 13463.754} C_VEL
LIN {X 0,Y 402.85,Z 714.051,A -85,B 0,C 180,E1 13461.532,E2 13461.532} C_VEL
LIN {X 0,Y 400.027,Z 728.131,A -85,B 0,C 180,E1 13459.013,E2 13459.013} C_VEL
LIN {X 0,Y 397.666,Z 740.259,A -85,B 0,C 180,E1 13456.397,E2 13456.397} C_VEL
LIN {X 0,Y 395.818,Z 750.451,A -85,B 0,C 180,E1 13453.745,E2 13453.745} C_VEL
LIN {X 0,Y 394.341,Z 759.486,A -85,B 0,C 180,E1 13450.858,E2 13450.858} C_VEL
LIN {X 0,Y 393.337,Z 766.608,A -85,B 0,C 180,E1 13447.965,E2 13447.965} C_VEL
LIN {X 0,Y 392.731,Z 771.954,A -85,B 0,C 180,E1 13445.127,E2 13445.127} C_VEL
LIN {X 0,Y 392.387,Z 776.101,A -85,B 0,C 180,E1 13442.008,E2 13442.008} C_VEL
LIN {X 0,Y 392.249,Z 778.446,A -85,B 0,C 180,E1 13439.039,E2 13439.039} C_VEL
LIN {X 0,Y 392.212,Z 779.22,A -85,B 0,C 180,E1 13436.171,E2 13436.171} C_VEL
LIN {X 0,Y 392.204,Z 779.192,A -85,B 0,C 180,E1 13435.624,E2 13435.624} C_VEL
LIN {X 0,Y 391.215,Z 779.103,A -85,B 0,C 180,E1 13434.498,E2 13434.498} C_VEL
LIN {X 0,Y 384.96,Z 778.074,A -85,B 0,C 180,E1 13431.407,E2 13431.407} C_VEL
LIN {X 0,Y 384.362,Z 777.3,A -85,B 0,C 180,E1 13430.504,E2 13430.504} C_VEL
LIN {X 0,Y 384.655,Z 773.548,A -85,B 0,C 180,E1 13427.395,E2 13427.395} C_VEL
LIN {X 0,Y 385.241,Z 767.978,A -85,B 0,C 180,E1 13424.276,E2 13424.276} C_VEL
LIN {X 0,Y 386.178,Z 761.038,A -85,B 0,C 180,E1 13421.35,E2 13421.35} C_VEL
LIN {X 0,Y 387.572,Z 752.399,A -85,B 0,C 180,E1 13418.457,E2 13418.457} C_VEL
LIN {X 0,Y 389.38,Z 742.491,A -85,B 0,C 180,E1 13415.749,E2 13415.749} C_VEL
LIN {X 0,Y 391.705,Z 730.658,A -85,B 0,C 180,E1 13413.074,E2 13413.074} C_VEL
LIN {X 0,Y 394.402,Z 717.373,A -85,B 0,C 180,E1 13410.583,E2 13410.583} C_VEL
LIN {X 0,Y 397.389,Z 702.572,A -85,B 0,C 180,E1 13408.271,E2 13408.271} C_VEL
LIN {X 0,Y 400.363,Z 687.358,A -85,B 0,C 180,E1 13406.279,E2 13406.279} C_VEL
LIN {X 0,Y 403.574,Z 670.063,A -85,B 0,C 180,E1 13404.386,E2 13404.386} C_VEL
LIN {X 0,Y 406.55,Z 652.563,A -85,B 0,C 180,E1 13402.796,E2 13402.796} C_VEL
LIN {X 0,Y 409.34,Z 634.309,A -85,B 0,C 180,E1 13401.433,E2 13401.433} C_VEL
LIN {X 0,Y 411.865,Z 614.589,A -85,B 0,C 180,E1 13400.26,E2 13400.26} C_VEL
LIN {X 0,Y 413.945,Z 594.379,A -85,B 0,C 180,E1 13399.331,E2 13399.331} C_VEL
LIN {X 0,Y 415.581,Z 573.533,A -85,B 0,C 180,E1 13398.636,E2 13398.636} C_VEL
LIN {X 0,Y 416.811,Z 546.799,A -85,B 0,C 180,E1 13398.057,E2 13398.057} C_VEL
LIN {X 0,Y 424.388,Z 339.114,A -85,B 0,C 180,E1 13394.159,E2 13394.159} C_VEL
LIN {X 0,Y 423.471,Z 334.486,A -85,B 0,C 180,E1 13393.932,E2 13393.932} C_VEL
LIN {X 0,Y 412.224,Z 315.459,A -85,B 0,C 180,E1 13391.947,E2 13391.947} C_VEL
LIN {X 0,Y 402.099,Z 299.629,A -85,B 0,C 180,E1 13390.035,E2 13390.035} C_VEL
LIN {X 0,Y 395.701,Z 285.564,A -85,B 0,C 180,E1 13387.102,E2 13387.102} C_VEL
LIN {X 0,Y 391.548,Z 277.101,A -85,B 0,C 180,E1 13385.163,E2 13385.163} C_VEL
LIN {X 0,Y 389.357,Z 272.788,A -85,B 0,C 180,E1 13384.118,E2 13384.118} C_VEL
LIN {X 0,Y 387.431,Z 268.871,A -85,B 0,C 180,E1 13383.154,E2 13383.154} C_VEL
LIN {X 0,Y 385.748,Z 265.405,A -85,B 0,C 180,E1 13382.275,E2 13382.275} C_VEL
LIN {X 0,Y 385.631,Z 264.695,A -85,B 0,C 180,E1 13381.825,E2 13381.825} C_VEL
LIN {X 0,Y 385.623,Z 264.683,A -85,B 0,C 180,E1 13377.893,E2 13377.893} C_VEL
LIN {X 0,Y 385.621,Z 264.682,A -85,B 0,C 180,E1 13373.946,E2 13373.946} C_VEL
LIN {X 0,Y 385.625,Z 264.679,A -85,B 0,C 180,E1 13369.894,E2 13369.894} C_VEL
LIN {X 0,Y 385.623,Z 264.678,A -85,B 0,C 180,E1 13365.905,E2 13365.905} C_VEL
LIN {X 0,Y 385.623,Z 264.682,A -85,B 0,C 180,E1 13361.917,E2 13361.917} C_VEL
LIN {X 0,Y 385.627,Z 264.696,A -85,B 0,C 180,E1 13357.913,E2 13357.913} C_VEL
LIN {X 0,Y 385.626,Z 264.695,A -85,B 0,C 180,E1 13353.878,E2 13353.878} C_VEL
LIN {X 0,Y 385.629,Z 264.676,A -85,B 0,C 180,E1 13349.854,E2 13349.854} C_VEL
LIN {X 0,Y 385.62,Z 264.676,A -85,B 0,C 180,E1 13345.822,E2 13345.822} C_VEL
LIN {X 0,Y 385.632,Z 264.698,A -85,B 0,C 180,E1 13341.761,E2 13341.761} C_VEL
LIN {X 0,Y 385.623,Z 264.693,A -85,B 0,C 180,E1 13337.658,E2 13337.658} C_VEL
LIN {X 0,Y 385.623,Z 264.669,A -85,B 0,C 180,E1 13333.646,E2 13333.646} C_VEL
LIN {X 0,Y 385.62,Z 264.682,A -85,B 0,C 180,E1 13329.551,E2 13329.551} C_VEL
LIN {X 0,Y 385.623,Z 264.701,A -85,B 0,C 180,E1 13325.504,E2 13325.504} C_VEL
LIN {X 0,Y 385.621,Z 264.686,A -85,B 0,C 180,E1 13321.485,E2 13321.485} C_VEL
LIN {X 0,Y 385.616,Z 264.673,A -85,B 0,C 180,E1 13317.472,E2 13317.472} C_VEL
LIN {X 0,Y 385.618,Z 264.682,A -85,B 0,C 180,E1 13313.448,E2 13313.448} C_VEL
LIN {X 0,Y 385.616,Z 264.698,A -85,B 0,C 180,E1 13309.391,E2 13309.391} C_VEL
LIN {X 0,Y 385.624,Z 264.701,A -85,B 0,C 180,E1 13305.279,E2 13305.279} C_VEL
LIN {X 0,Y 385.622,Z 264.7,A -85,B 0,C 180,E1 13301.147,E2 13301.147} C_VEL
LIN {X 0,Y 385.625,Z 264.7,A -85,B 0,C 180,E1 13297.112,E2 13297.112} C_VEL
LIN {X 0,Y 385.623,Z 264.703,A -85,B 0,C 180,E1 13293.015,E2 13293.015} C_VEL
LIN {X 0,Y 385.629,Z 264.925,A -85,B 0,C 180,E1 13289.628,E2 13289.628} C_VEL
LIN {X 0,Y 387.147,Z 268.473,A -85,B 0,C 180,E1 13288.727,E2 13288.727} C_VEL
LIN {X 0,Y 388.249,Z 269.909,A -85,B 0,C 180,E1 13288.307,E2 13288.307} C_VEL
LIN {X 0,Y 390.1,Z 273.686,A -85,B 0,C 180,E1 13287.435,E2 13287.435} C_VEL
LIN {X 0,Y 395.504,Z 283.648,A -85,B 0,C 180,E1 13285.155,E2 13285.155} C_VEL
LIN {X 0,Y 403.544,Z 299.687,A -85,B 0,C 180,E1 13281.906,E2 13281.906} C_VEL
LIN {X 0,Y 405.258,Z 302.933,A -85,B 0,C 180,E1 13281.398,E2 13281.398} C_VEL
LIN {X 0,Y 416.831,Z 320.44,A -85,B 0,C 180,E1 13279.25,E2 13279.25} C_VEL
LIN {X 0,Y 428.873,Z 340.358,A -85,B 0,C 180,E1 13277.165,E2 13277.165} C_VEL
LIN {X 0,Y 428.932,Z 345.789,A -85,B 0,C 180,E1 13277.032,E2 13277.032} C_VEL
LIN {X 0,Y 421.735,Z 559.211,A -85,B 0,C 180,E1 13273.127,E2 13273.127} C_VEL
LIN {X 0,Y 420.102,Z 604.979,A -85,B 0,C 180,E1 13272.261,E2 13272.261} C_VEL
LIN {X 0,Y 418.285,Z 627.094,A -85,B 0,C 180,E1 13271.632,E2 13271.632} C_VEL
LIN {X 0,Y 416.001,Z 648.177,A -85,B 0,C 180,E1 13270.79,E2 13270.79} C_VEL
LIN {X 0,Y 413.259,Z 669.261,A -85,B 0,C 180,E1 13269.695,E2 13269.695} C_VEL
LIN {X 0,Y 410.248,Z 688.869,A -85,B 0,C 180,E1 13268.422,E2 13268.422} C_VEL
LIN {X 0,Y 406.902,Z 708.188,A -85,B 0,C 180,E1 13266.885,E2 13266.885} C_VEL
LIN {X 0,Y 403.316,Z 727.626,A -85,B 0,C 180,E1 13265.021,E2 13265.021} C_VEL
LIN {X 0,Y 399.817,Z 745.517,A -85,B 0,C 180,E1 13262.983,E2 13262.983} C_VEL
LIN {X 0,Y 396.424,Z 762.485,A -85,B 0,C 180,E1 13260.675,E2 13260.675} C_VEL
LIN {X 0,Y 393.352,Z 777.861,A -85,B 0,C 180,E1 13258.214,E2 13258.214} C_VEL
LIN {X 0,Y 390.721,Z 791.705,A -85,B 0,C 180,E1 13255.623,E2 13255.623} C_VEL
LIN {X 0,Y 388.508,Z 804.202,A -85,B 0,C 180,E1 13252.866,E2 13252.866} C_VEL
LIN {X 0,Y 386.766,Z 815.33,A -85,B 0,C 180,E1 13249.951,E2 13249.951} C_VEL
LIN {X 0,Y 385.468,Z 825.275,A -85,B 0,C 180,E1 13246.834,E2 13246.834} C_VEL
LIN {X 0,Y 384.678,Z 833.074,A -85,B 0,C 180,E1 13243.833,E2 13243.833} C_VEL
LIN {X 0,Y 384.257,Z 839.275,A -85,B 0,C 180,E1 13240.796,E2 13240.796} C_VEL
LIN {X 0,Y 384.073,Z 843.978,A -85,B 0,C 180,E1 13237.778,E2 13237.778} C_VEL
LIN {X 0,Y 384.048,Z 847.013,A -85,B 0,C 180,E1 13234.777,E2 13234.777} C_VEL
LIN {X 0,Y 384.053,Z 848.691,A -85,B 0,C 180,E1 13231.639,E2 13231.639} C_VEL
LIN {X 0,Y 384.063,Z 848.742,A -85,B 0,C 180,E1 13228.805,E2 13228.805} C_VEL
LIN {X 0,Y 384.05,Z 847.285,A -85,B 0,C 180,E1 13225.657,E2 13225.657} C_VEL
LIN {X 0,Y 384.082,Z 844.53,A -85,B 0,C 180,E1 13222.82,E2 13222.82} C_VEL
LIN {X 0,Y 384.229,Z 839.831,A -85,B 0,C 180,E1 13219.627,E2 13219.627} C_VEL
LIN {X 0,Y 384.596,Z 833.855,A -85,B 0,C 180,E1 13216.62,E2 13216.62} C_VEL
LIN {X 0,Y 385.328,Z 826.04,A -85,B 0,C 180,E1 13213.569,E2 13213.569} C_VEL
LIN {X 0,Y 386.515,Z 816.472,A -85,B 0,C 180,E1 13210.505,E2 13210.505} C_VEL
LIN {X 0,Y 388.157,Z 805.523,A -85,B 0,C 180,E1 13207.588,E2 13207.588} C_VEL
LIN {X 0,Y 390.254,Z 793.18,A -85,B 0,C 180,E1 13204.829,E2 13204.829} C_VEL
LIN {X 0,Y 392.939,Z 778.771,A -85,B 0,C 180,E1 13202.081,E2 13202.081} C_VEL
LIN {X 0,Y 395.962,Z 763.386,A -85,B 0,C 180,E1 13199.582,E2 13199.582} C_VEL
LIN {X 0,Y 399.289,Z 746.392,A -85,B 0,C 180,E1 13197.255,E2 13197.255} C_VEL
LIN {X 0,Y 402.786,Z 728.514,A -85,B 0,C 180,E1 13195.183,E2 13195.183} C_VEL
LIN {X 0,Y 406.252,Z 709.874,A -85,B 0,C 180,E1 13193.355,E2 13193.355} C_VEL
LIN {X 0,Y 409.634,Z 690.463,A -85,B 0,C 180,E1 13191.773,E2 13191.773} C_VEL
LIN {X 0,Y 412.623,Z 671.361,A -85,B 0,C 180,E1 13190.498,E2 13190.498} C_VEL
LIN {X 0,Y 415.446,Z 650.789,A -85,B 0,C 180,E1 13189.381,E2 13189.381} C_VEL
LIN {X 0,Y 417.83,Z 629.741,A -85,B 0,C 180,E1 13188.498,E2 13188.498} C_VEL
LIN {X 0,Y 419.709,Z 608.027,A -85,B 0,C 180,E1 13187.844,E2 13187.844} C_VEL
LIN {X 0,Y 421.019,Z 578.64,A -85,B 0,C 180,E1 13187.243,E2 13187.243} C_VEL
LIN {X 0,Y 428.244,Z 367.036,A -85,B 0,C 180,E1 13183.353,E2 13183.353} C_VEL
LIN {X 0,Y 429.047,Z 340.77,A -85,B 0,C 180,E1 13182.836,E2 13182.836} C_VEL
LIN {X 0,Y 428.352,Z 338.842,A -85,B 0,C 180,E1 13182.695,E2 13182.695} C_VEL
LIN {X 0,Y 417.789,Z 320.785,A -85,B 0,C 180,E1 13180.705,E2 13180.705} C_VEL
LIN {X 0,Y 408.065,Z 305.818,A -85,B 0,C 180,E1 13178.714,E2 13178.714} C_VEL
LIN {X 0,Y 404.857,Z 300.915,A -85,B 0,C 180,E1 13177.949,E2 13177.949} C_VEL
LIN {X 0,Y 398.749,Z 288.753,A -85,B 0,C 180,E1 13175.169,E2 13175.169} C_VEL
LIN {X 0,Y 395.781,Z 283.436,A -85,B 0,C 180,E1 13173.766,E2 13173.766} C_VEL
LIN {X 0,Y 393.831,Z 279.602,A -85,B 0,C 180,E1 13172.737,E2 13172.737} C_VEL
LIN {X 0,Y 391.681,Z 275.567,A -85,B 0,C 180,E1 13171.555,E2 13171.555} C_VEL
LIN {X 0,Y 389.184,Z 271.677,A -85,B 0,C 180,E1 13170.236,E2 13170.236} C_VEL
LIN {X 0,Y 388.29,Z 269.732,A -85,B 0,C 180,E1 13169.631,E2 13169.631} C_VEL
LIN {X 0,Y 386.181,Z 266.798,A -85,B 0,C 180,E1 13168.451,E2 13168.451} C_VEL
LIN {X 0,Y 385.663,Z 264.966,A -85,B 0,C 180,E1 13167.819,E2 13167.819} C_VEL
LIN {X 0,Y 385.622,Z 264.691,A -85,B 0,C 180,E1 13164.022,E2 13164.022} C_VEL
LIN {X 0,Y 385.622,Z 264.69,A -85,B 0,C 180,E1 13160.015,E2 13160.015} C_VEL
LIN {X 0,Y 385.622,Z 264.701,A -85,B 0,C 180,E1 13155.954,E2 13155.954} C_VEL
LIN {X 0,Y 385.62,Z 264.694,A -85,B 0,C 180,E1 13151.973,E2 13151.973} C_VEL
LIN {X 0,Y 385.621,Z 264.688,A -85,B 0,C 180,E1 13147.9,E2 13147.9} C_VEL
LIN {X 0,Y 385.612,Z 264.692,A -85,B 0,C 180,E1 13143.867,E2 13143.867} C_VEL
LIN {X 0,Y 385.617,Z 264.703,A -85,B 0,C 180,E1 13139.853,E2 13139.853} C_VEL
LIN {X 0,Y 385.61,Z 264.692,A -85,B 0,C 180,E1 13135.838,E2 13135.838} C_VEL
LIN {X 0,Y 385.634,Z 265.005,A -85,B 0,C 180,E1 13133.451,E2 13133.451} C_VEL
LIN {X 0,Y 387.201,Z 268.549,A -85,B 0,C 180,E1 13132.135,E2 13132.135} C_VEL
LIN {X 0,Y 388.666,Z 270.682,A -85,B 0,C 180,E1 13131.271,E2 13131.271} C_VEL
LIN {X 0,Y 390.758,Z 274.454,A -85,B 0,C 180,E1 13129.981,E2 13129.981} C_VEL
LIN {X 0,Y 393.869,Z 280.393,A -85,B 0,C 180,E1 13128.135,E2 13128.135} C_VEL
LIN {X 0,Y 398.225,Z 288.874,A -85,B 0,C 180,E1 13125.757,E2 13125.757} C_VEL
LIN {X 0,Y 403.584,Z 300.266,A -85,B 0,C 180,E1 13123.003,E2 13123.003} C_VEL
LIN {X 0,Y 414.191,Z 316.41,A -85,B 0,C 180,E1 13120.667,E2 13120.667} C_VEL
LIN {X 0,Y 424.344,Z 333.163,A -85,B 0,C 180,E1 13118.653,E2 13118.653} C_VEL
LIN {X 0,Y 426.683,Z 337.717,A -85,B 0,C 180,E1 13118.199,E2 13118.199} C_VEL
LIN {X 0,Y 426.973,Z 341.699,A -85,B 0,C 180,E1 13118.055,E2 13118.055} C_VEL
LIN {X 0,Y 417.349,Z 569.97,A -85,B 0,C 180,E1 13113.629,E2 13113.629} C_VEL
LIN {X 0,Y 415.783,Z 590.742,A -85,B 0,C 180,E1 13112.981,E2 13112.981} C_VEL
LIN {X 0,Y 413.729,Z 610.629,A -85,B 0,C 180,E1 13112.119,E2 13112.119} C_VEL
LIN {X 0,Y 411.22,Z 630.344,A -85,B 0,C 180,E1 13111.006,E2 13111.006} C_VEL
LIN {X 0,Y 408.377,Z 649.118,A -85,B 0,C 180,E1 13109.677,E2 13109.677} C_VEL
LIN {X 0,Y 405.32,Z 666.873,A -85,B 0,C 180,E1 13108.138,E2 13108.138} C_VEL
LIN {X 0,Y 402.054,Z 684.072,A -85,B 0,C 180,E1 13106.321,E2 13106.321} C_VEL
LIN {X 0,Y 398.823,Z 699.855,A -85,B 0,C 180,E1 13104.321,E2 13104.321} C_VEL
LIN {X 0,Y 395.758,Z 714.367,A -85,B 0,C 180,E1 13102.128,E2 13102.128} C_VEL
LIN {X 0,Y 392.88,Z 727.91,A -85,B 0,C 180,E1 13099.687,E2 13099.687} C_VEL
LIN {X 0,Y 390.385,Z 739.903,A -85,B 0,C 180,E1 13097.098,E2 13097.098} C_VEL
LIN {X 0,Y 388.259,Z 750.755,A -85,B 0,C 180,E1 13094.259,E2 13094.259} C_VEL
LIN {X 0,Y 386.612,Z 759.996,A -85,B 0,C 180,E1 13091.262,E2 13091.262} C_VEL
LIN {X 0,Y 385.511,Z 767.165,A -85,B 0,C 180,E1 13088.308,E2 13088.308} C_VEL
LIN {X 0,Y 384.825,Z 772.678,A -85,B 0,C 180,E1 13085.333,E2 13085.333} C_VEL
LIN {X 0,Y 384.449,Z 776.752,A -85,B 0,C 180,E1 13082.22,E2 13082.22} C_VEL
LIN {X 0,Y 384.291,Z 779.099,A -85,B 0,C 180,E1 13079.286,E2 13079.286} C_VEL
LIN {X 0,Y 384.244,Z 779.928,A -85,B 0,C 180,E1 13076.256,E2 13076.256} C_VEL
LIN {X 0,Y 384.258,Z 779.245,A -85,B 0,C 180,E1 13073.294,E2 13073.294} C_VEL
LIN {X 0,Y 384.362,Z 777.3,A -85,B 0,C 180,E1 13070.504,E2 13070.504} C_VEL
LIN {X 0,Y 383.444,Z 776.226,A -85,B 0,C 180,E1 13069.365,E2 13069.365} C_VEL
LIN {X 0,Y 377.617,Z 772.841,A -85,B 0,C 180,E1 13066.322,E2 13066.322} C_VEL
LIN {X 0,Y 377.059,Z 771.189,A -85,B 0,C 180,E1 13065.342,E2 13065.342} C_VEL
LIN {X 0,Y 377.94,Z 764.698,A -85,B 0,C 180,E1 13062.22,E2 13062.22} C_VEL
LIN {X 0,Y 379.227,Z 756.726,A -85,B 0,C 180,E1 13059.257,E2 13059.257} C_VEL
LIN {X 0,Y 381.047,Z 746.956,A -85,B 0,C 180,E1 13056.329,E2 13056.329} C_VEL
LIN {X 0,Y 383.308,Z 735.825,A -85,B 0,C 180,E1 13053.591,E2 13053.591} C_VEL
LIN {X 0,Y 385.991,Z 723.232,A -85,B 0,C 180,E1 13051.015,E2 13051.015} C_VEL
LIN {X 0,Y 388.931,Z 709.589,A -85,B 0,C 180,E1 13048.676,E2 13048.676} C_VEL
LIN {X 0,Y 392.25,Z 693.783,A -85,B 0,C 180,E1 13046.422,E2 13046.422} C_VEL
LIN {X 0,Y 395.47,Z 677.502,A -85,B 0,C 180,E1 13044.488,E2 13044.488} C_VEL
LIN {X 0,Y 398.731,Z 659.805,A -85,B 0,C 180,E1 13042.741,E2 13042.741} C_VEL
LIN {X 0,Y 401.88,Z 640.751,A -85,B 0,C 180,E1 13041.2,E2 13041.2} C_VEL
LIN {X 0,Y 404.585,Z 621.862,A -85,B 0,C 180,E1 13039.968,E2 13039.968} C_VEL
LIN {X 0,Y 406.959,Z 601.911,A -85,B 0,C 180,E1 13038.944,E2 13038.944} C_VEL
LIN {X 0,Y 408.869,Z 580.713,A -85,B 0,C 180,E1 13038.139,E2 13038.139} C_VEL
LIN {X 0,Y 410.139,Z 559.475,A -85,B 0,C 180,E1 13037.596,E2 13037.596} C_VEL
LIN {X 0,Y 418.564,Z 340.833,A -85,B 0,C 180,E1 13033.442,E2 13033.442} C_VEL
LIN {X 0,Y 417.973,Z 338.435,A -85,B 0,C 180,E1 13033.305,E2 13033.305} C_VEL
LIN {X 0,Y 407.277,Z 320.338,A -85,B 0,C 180,E1 13031.368,E2 13031.368} C_VEL
LIN {X 0,Y 396.469,Z 303.497,A -85,B 0,C 180,E1 13029.273,E2 13029.273} C_VEL
LIN {X 0,Y 393.877,Z 299.317,A -85,B 0,C 180,E1 13028.685,E2 13028.685} C_VEL
LIN {X 0,Y 386.593,Z 283.605,A -85,B 0,C 180,E1 13025.198,E2 13025.198} C_VEL
LIN {X 0,Y 381.856,Z 274.428,A -85,B 0,C 180,E1 13022.898,E2 13022.898} C_VEL
LIN {X 0,Y 379.419,Z 269.736,A -85,B 0,C 180,E1 13021.658,E2 13021.658} C_VEL
LIN {X 0,Y 377.87,Z 266.698,A -85,B 0,C 180,E1 13020.828,E2 13020.828} C_VEL
LIN {X 0,Y 377.69,Z 265.705,A -85,B 0,C 180,E1 13020.417,E2 13020.417} C_VEL
LIN {X 0,Y 377.685,Z 265.691,A -85,B 0,C 180,E1 13016.409,E2 13016.409} C_VEL
LIN {X 0,Y 377.685,Z 265.691,A -85,B 0,C 180,E1 13012.302,E2 13012.302} C_VEL
LIN {X 0,Y 377.688,Z 265.689,A -85,B 0,C 180,E1 13008.157,E2 13008.157} C_VEL
LIN {X 0,Y 377.685,Z 265.684,A -85,B 0,C 180,E1 13004.124,E2 13004.124} C_VEL
LIN {X 0,Y 377.687,Z 265.668,A -85,B 0,C 180,E1 13000.036,E2 13000.036} C_VEL
LIN {X 0,Y 377.679,Z 265.661,A -85,B 0,C 180,E1 12995.993,E2 12995.993} C_VEL
LIN {X 0,Y 377.683,Z 265.672,A -85,B 0,C 180,E1 12991.968,E2 12991.968} C_VEL
LIN {X 0,Y 377.694,Z 265.688,A -85,B 0,C 180,E1 12987.853,E2 12987.853} C_VEL
LIN {X 0,Y 377.687,Z 265.677,A -85,B 0,C 180,E1 12983.661,E2 12983.661} C_VEL
LIN {X 0,Y 377.682,Z 265.659,A -85,B 0,C 180,E1 12979.645,E2 12979.645} C_VEL
LIN {X 0,Y 377.688,Z 265.672,A -85,B 0,C 180,E1 12975.507,E2 12975.507} C_VEL
LIN {X 0,Y 377.685,Z 265.686,A -85,B 0,C 180,E1 12971.451,E2 12971.451} C_VEL
LIN {X 0,Y 377.688,Z 265.667,A -85,B 0,C 180,E1 12967.299,E2 12967.299} C_VEL
LIN {X 0,Y 377.682,Z 265.662,A -85,B 0,C 180,E1 12963.186,E2 12963.186} C_VEL
LIN {X 0,Y 377.687,Z 265.676,A -85,B 0,C 180,E1 12959.089,E2 12959.089} C_VEL
LIN {X 0,Y 377.686,Z 265.688,A -85,B 0,C 180,E1 12954.987,E2 12954.987} C_VEL
LIN {X 0,Y 377.685,Z 265.678,A -85,B 0,C 180,E1 12950.9,E2 12950.9} C_VEL
LIN {X 0,Y 377.686,Z 265.666,A -85,B 0,C 180,E1 12946.839,E2 12946.839} C_VEL
LIN {X 0,Y 377.683,Z 265.667,A -85,B 0,C 180,E1 12942.751,E2 12942.751} C_VEL
LIN {X 0,Y 377.69,Z 265.667,A -85,B 0,C 180,E1 12938.719,E2 12938.719} C_VEL
LIN {X 0,Y 377.683,Z 265.67,A -85,B 0,C 180,E1 12934.603,E2 12934.603} C_VEL
LIN {X 0,Y 377.711,Z 265.934,A -85,B 0,C 180,E1 12931.184,E2 12931.184} C_VEL
LIN {X 0,Y 379.132,Z 269.375,A -85,B 0,C 180,E1 12930.277,E2 12930.277} C_VEL
LIN {X 0,Y 380.492,Z 271.389,A -85,B 0,C 180,E1 12929.698,E2 12929.698} C_VEL
LIN {X 0,Y 382.74,Z 275.33,A -85,B 0,C 180,E1 12928.676,E2 12928.676} C_VEL
LIN {X 0,Y 390.246,Z 289.731,A -85,B 0,C 180,E1 12925.333,E2 12925.333} C_VEL
LIN {X 0,Y 396.593,Z 302.132,A -85,B 0,C 180,E1 12922.79,E2 12922.79} C_VEL
LIN {X 0,Y 410.49,Z 323.017,A -85,B 0,C 180,E1 12920.094,E2 12920.094} C_VEL
LIN {X 0,Y 423.218,Z 344.052,A -85,B 0,C 180,E1 12917.813,E2 12917.813} C_VEL
LIN {X 0,Y 415.781,Z 553.974,A -85,B 0,C 180,E1 12913.93,E2 12913.93} C_VEL
LIN {X 0,Y 413.926,Z 604.417,A -85,B 0,C 180,E1 12912.969,E2 12912.969} C_VEL
LIN {X 0,Y 412.043,Z 626.556,A -85,B 0,C 180,E1 12912.335,E2 12912.335} C_VEL
LIN {X 0,Y 409.661,Z 647.608,A -85,B 0,C 180,E1 12911.49,E2 12911.49} C_VEL
LIN {X 0,Y 406.825,Z 668.573,A -85,B 0,C 180,E1 12910.394,E2 12910.394} C_VEL
LIN {X 0,Y 403.787,Z 687.553,A -85,B 0,C 180,E1 12909.153,E2 12909.153} C_VEL
LIN {X 0,Y 400.196,Z 707.489,A -85,B 0,C 180,E1 12907.559,E2 12907.559} C_VEL
LIN {X 0,Y 396.497,Z 726.654,A -85,B 0,C 180,E1 12905.708,E2 12905.708} C_VEL
LIN {X 0,Y 392.891,Z 744.337,A -85,B 0,C 180,E1 12903.677,E2 12903.677} C_VEL
LIN {X 0,Y 389.282,Z 761.347,A -85,B 0,C 180,E1 12901.338,E2 12901.338} C_VEL
LIN {X 0,Y 385.987,Z 776.995,A -85,B 0,C 180,E1 12898.802,E2 12898.802} C_VEL
LIN {X 0,Y 383.188,Z 790.933,A -85,B 0,C 180,E1 12896.154,E2 12896.154} C_VEL
LIN {X 0,Y 380.838,Z 803.414,A -85,B 0,C 180,E1 12893.354,E2 12893.354} C_VEL
LIN {X 0,Y 378.975,Z 814.564,A -85,B 0,C 180,E1 12890.379,E2 12890.379} C_VEL
LIN {X 0,Y 377.603,Z 824.383,A -85,B 0,C 180,E1 12887.25,E2 12887.25} C_VEL
LIN {X 0,Y 376.736,Z 832.337,A -85,B 0,C 180,E1 12884.131,E2 12884.131} C_VEL
LIN {X 0,Y 376.281,Z 838.551,A -85,B 0,C 180,E1 12881.028,E2 12881.028} C_VEL
LIN {X 0,Y 376.096,Z 843.263,A -85,B 0,C 180,E1 12877.944,E2 12877.944} C_VEL
LIN {X 0,Y 376.074,Z 846.301,A -85,B 0,C 180,E1 12874.879,E2 12874.879} C_VEL
LIN {X 0,Y 376.083,Z 847.956,A -85,B 0,C 180,E1 12871.827,E2 12871.827} C_VEL
LIN {X 0,Y 376.096,Z 848.051,A -85,B 0,C 180,E1 12868.932,E2 12868.932} C_VEL
LIN {X 0,Y 376.075,Z 846.811,A -85,B 0,C 180,E1 12865.882,E2 12865.882} C_VEL
LIN {X 0,Y 376.101,Z 843.965,A -85,B 0,C 180,E1 12862.821,E2 12862.821} C_VEL
LIN {X 0,Y 376.249,Z 839.248,A -85,B 0,C 180,E1 12859.501,E2 12859.501} C_VEL
LIN {X 0,Y 376.619,Z 833.412,A -85,B 0,C 180,E1 12856.488,E2 12856.488} C_VEL
LIN {X 0,Y 377.383,Z 825.681,A -85,B 0,C 180,E1 12853.371,E2 12853.371} C_VEL
LIN {X 0,Y 378.629,Z 816.199,A -85,B 0,C 180,E1 12850.243,E2 12850.243} C_VEL
LIN {X 0,Y 380.349,Z 805.303,A -85,B 0,C 180,E1 12847.266,E2 12847.266} C_VEL
LIN {X 0,Y 382.639,Z 792.625,A -85,B 0,C 180,E1 12844.358,E2 12844.358} C_VEL
LIN {X 0,Y 385.478,Z 778.241,A -85,B 0,C 180,E1 12841.559,E2 12841.559} C_VEL
LIN {X 0,Y 388.659,Z 762.996,A -85,B 0,C 180,E1 12839.033,E2 12839.033} C_VEL
LIN {X 0,Y 392.159,Z 746.055,A -85,B 0,C 180,E1 12836.67,E2 12836.67} C_VEL
LIN {X 0,Y 395.829,Z 728.238,A -85,B 0,C 180,E1 12834.568,E2 12834.568} C_VEL
LIN {X 0,Y 399.467,Z 709.703,A -85,B 0,C 180,E1 12832.718,E2 12832.718} C_VEL
LIN {X 0,Y 403.01,Z 690.37,A -85,B 0,C 180,E1 12831.119,E2 12831.119} C_VEL
LIN {X 0,Y 406.128,Z 671.397,A -85,B 0,C 180,E1 12829.831,E2 12829.831} C_VEL
LIN {X 0,Y 409.071,Z 651.009,A -85,B 0,C 180,E1 12828.703,E2 12828.703} C_VEL
LIN {X 0,Y 411.608,Z 629.642,A -85,B 0,C 180,E1 12827.795,E2 12827.795} C_VEL
LIN {X 0,Y 413.59,Z 607.941,A -85,B 0,C 180,E1 12827.131,E2 12827.131} C_VEL
LIN {X 0,Y 414.909,Z 580.734,A -85,B 0,C 180,E1 12826.559,E2 12826.559} C_VEL
LIN {X 0,Y 422.402,Z 372.783,A -85,B 0,C 180,E1 12822.69,E2 12822.69} C_VEL
LIN {X 0,Y 423.418,Z 343.55,A -85,B 0,C 180,E1 12822.117,E2 12822.117} C_VEL
LIN {X 0,Y 413.202,Z 325.867,A -85,B 0,C 180,E1 12820.116,E2 12820.116} C_VEL
LIN {X 0,Y 403.783,Z 311.295,A -85,B 0,C 180,E1 12818.113,E2 12818.113} C_VEL
LIN {X 0,Y 396.857,Z 301.22,A -85,B 0,C 180,E1 12816.484,E2 12816.484} C_VEL
LIN {X 0,Y 391.471,Z 290.472,A -85,B 0,C 180,E1 12813.835,E2 12813.835} C_VEL
LIN {X 0,Y 388.592,Z 285.314,A -85,B 0,C 180,E1 12812.358,E2 12812.358} C_VEL
LIN {X 0,Y 386.194,Z 280.876,A -85,B 0,C 180,E1 12811.013,E2 12811.013} C_VEL
LIN {X 0,Y 384.168,Z 277.252,A -85,B 0,C 180,E1 12809.81,E2 12809.81} C_VEL
LIN {X 0,Y 383.433,Z 275.964,A -85,B 0,C 180,E1 12809.357,E2 12809.357} C_VEL
LIN {X 0,Y 381.248,Z 272.427,A -85,B 0,C 180,E1 12807.999,E2 12807.999} C_VEL
LIN {X 0,Y 380.422,Z 270.785,A -85,B 0,C 180,E1 12807.385,E2 12807.385} C_VEL
LIN {X 0,Y 378.156,Z 267.57,A -85,B 0,C 180,E1 12805.867,E2 12805.867} C_VEL
LIN {X 0,Y 377.707,Z 265.87,A -85,B 0,C 180,E1 12805.129,E2 12805.129} C_VEL
LIN {X 0,Y 377.68,Z 265.679,A -85,B 0,C 180,E1 12801.104,E2 12801.104} C_VEL
LIN {X 0,Y 377.674,Z 265.678,A -85,B 0,C 180,E1 12797.09,E2 12797.09} C_VEL
LIN {X 0,Y 377.675,Z 265.687,A -85,B 0,C 180,E1 12793.027,E2 12793.027} C_VEL
LIN {X 0,Y 377.669,Z 265.688,A -85,B 0,C 180,E1 12788.987,E2 12788.987} C_VEL
LIN {X 0,Y 377.663,Z 265.68,A -85,B 0,C 180,E1 12785.013,E2 12785.013} C_VEL
LIN {X 0,Y 377.662,Z 265.681,A -85,B 0,C 180,E1 12780.911,E2 12780.911} C_VEL
LIN {X 0,Y 377.66,Z 265.693,A -85,B 0,C 180,E1 12776.814,E2 12776.814} C_VEL
LIN {X 0,Y 377.725,Z 265.994,A -85,B 0,C 180,E1 12776.055,E2 12776.055} C_VEL
LIN {X 0,Y 379.193,Z 269.479,A -85,B 0,C 180,E1 12774.554,E2 12774.554} C_VEL
LIN {X 0,Y 380.807,Z 271.536,A -85,B 0,C 180,E1 12773.519,E2 12773.519} C_VEL
LIN {X 0,Y 382.581,Z 275.095,A -85,B 0,C 180,E1 12772.191,E2 12772.191} C_VEL
LIN {X 0,Y 383.744,Z 276.942,A -85,B 0,C 180,E1 12771.46,E2 12771.46} C_VEL
LIN {X 0,Y 386.442,Z 282.055,A -85,B 0,C 180,E1 12769.717,E2 12769.717} C_VEL
LIN {X 0,Y 388.818,Z 286.653,A -85,B 0,C 180,E1 12768.28,E2 12768.28} C_VEL
LIN {X 0,Y 392.873,Z 294.572,A -85,B 0,C 180,E1 12766.01,E2 12766.01} C_VEL
LIN {X 0,Y 395.825,Z 300.892,A -85,B 0,C 180,E1 12764.471,E2 12764.471} C_VEL
LIN {X 0,Y 404.291,Z 313.128,A -85,B 0,C 180,E1 12762.459,E2 12762.459} C_VEL
LIN {X 0,Y 414.172,Z 328.81,A -85,B 0,C 180,E1 12760.321,E2 12760.321} C_VEL
LIN {X 0,Y 421.472,Z 341.734,A -85,B 0,C 180,E1 12758.849,E2 12758.849} C_VEL
LIN {X 0,Y 411.495,Z 566.95,A -85,B 0,C 180,E1 12754.436,E2 12754.436} C_VEL
LIN {X 0,Y 409.983,Z 587.871,A -85,B 0,C 180,E1 12753.819,E2 12753.819} C_VEL
LIN {X 0,Y 407.845,Z 608.682,A -85,B 0,C 180,E1 12752.95,E2 12752.95} C_VEL
LIN {X 0,Y 405.367,Z 627.879,A -85,B 0,C 180,E1 12751.895,E2 12751.895} C_VEL
LIN {X 0,Y 402.463,Z 646.704,A -85,B 0,C 180,E1 12750.591,E2 12750.591} C_VEL
LIN {X 0,Y 399.263,Z 664.446,A -85,B 0,C 180,E1 12749.076,E2 12749.076} C_VEL
LIN {X 0,Y 395.865,Z 681.766,A -85,B 0,C 180,E1 12747.284,E2 12747.284} C_VEL
LIN {X 0,Y 392.261,Z 698.734,A -85,B 0,C 180,E1 12745.163,E2 12745.163} C_VEL
LIN {X 0,Y 389.03,Z 713.318,A -85,B 0,C 180,E1 12742.976,E2 12742.976} C_VEL
LIN {X 0,Y 385.959,Z 726.973,A -85,B 0,C 180,E1 12740.535,E2 12740.535} C_VEL
LIN {X 0,Y 383.159,Z 739.55,A -85,B 0,C 180,E1 12737.827,E2 12737.827} C_VEL
LIN {X 0,Y 380.813,Z 750.542,A -85,B 0,C 180,E1 12734.935,E2 12734.935} C_VEL
LIN {X 0,Y 379.077,Z 759.418,A -85,B 0,C 180,E1 12732.065,E2 12732.065} C_VEL
LIN {X 0,Y 377.811,Z 766.91,A -85,B 0,C 180,E1 12729.041,E2 12729.041} C_VEL
LIN {X 0,Y 376.985,Z 772.885,A -85,B 0,C 180,E1 12725.886,E2 12725.886} C_VEL
LIN {X 0,Y 376.548,Z 777.061,A -85,B 0,C 180,E1 12722.8,E2 12722.8} C_VEL
LIN {X 0,Y 376.347,Z 779.633,A -85,B 0,C 180,E1 12719.69,E2 12719.69} C_VEL
LIN {X 0,Y 376.277,Z 780.597,A -85,B 0,C 180,E1 12716.686,E2 12716.686} C_VEL
LIN {X 0,Y 376.287,Z 780.068,A -85,B 0,C 180,E1 12713.491,E2 12713.491} C_VEL
LIN {X 0,Y 376.404,Z 778.094,A -85,B 0,C 180,E1 12710.477,E2 12710.477} C_VEL
LIN {X 0,Y 376.694,Z 774.567,A -85,B 0,C 180,E1 12707.455,E2 12707.455} C_VEL
LIN {X 0,Y 377.059,Z 771.189,A -85,B 0,C 180,E1 12705.342,E2 12705.342} C_VEL
LIN {X 0,Y 376.334,Z 769.17,A -85,B 0,C 180,E1 12704.21,E2 12704.21} C_VEL
LIN {X 0,Y 371.152,Z 763.409,A -85,B 0,C 180,E1 12701.171,E2 12701.171} C_VEL
LIN {X 0,Y 370.839,Z 761.087,A -85,B 0,C 180,E1 12700.203,E2 12700.203} C_VEL
LIN {X 0,Y 372.502,Z 752.259,A -85,B 0,C 180,E1 12697.249,E2 12697.249} C_VEL
LIN {X 0,Y 374.64,Z 742.006,A -85,B 0,C 180,E1 12694.441,E2 12694.441} C_VEL
LIN {X 0,Y 377.347,Z 729.781,A -85,B 0,C 180,E1 12691.672,E2 12691.672} C_VEL
LIN {X 0,Y 380.249,Z 716.979,A -85,B 0,C 180,E1 12689.248,E2 12689.248} C_VEL
LIN {X 0,Y 383.632,Z 701.919,A -85,B 0,C 180,E1 12686.864,E2 12686.864} C_VEL
LIN {X 0,Y 387.237,Z 685.148,A -85,B 0,C 180,E1 12684.668,E2 12684.668} C_VEL
LIN {X 0,Y 390.667,Z 667.864,A -85,B 0,C 180,E1 12682.797,E2 12682.797} C_VEL
LIN {X 0,Y 393.836,Z 650.454,A -85,B 0,C 180,E1 12681.24,E2 12681.24} C_VEL
LIN {X 0,Y 396.897,Z 631.388,A -85,B 0,C 180,E1 12679.845,E2 12679.845} C_VEL
LIN {X 0,Y 399.515,Z 611.952,A -85,B 0,C 180,E1 12678.708,E2 12678.708} C_VEL
LIN {X 0,Y 401.783,Z 591.262,A -85,B 0,C 180,E1 12677.785,E2 12677.785} C_VEL
LIN {X 0,Y 403.432,Z 570.185,A -85,B 0,C 180,E1 12677.118,E2 12677.118} C_VEL
LIN {X 0,Y 405.271,Z 527.133,A -85,B 0,C 180,E1 12676.247,E2 12676.247} C_VEL
LIN {X 0,Y 412.715,Z 342.754,A -85,B 0,C 180,E1 12672.701,E2 12672.701} C_VEL
LIN {X 0,Y 401.659,Z 323.979,A -85,B 0,C 180,E1 12670.633,E2 12670.633} C_VEL
LIN {X 0,Y 389.351,Z 304.943,A -85,B 0,C 180,E1 12668.151,E2 12668.151} C_VEL
LIN {X 0,Y 385.575,Z 299.23,A -85,B 0,C 180,E1 12667.272,E2 12667.272} C_VEL
LIN {X 0,Y 380.401,Z 288.168,A -85,B 0,C 180,E1 12664.708,E2 12664.708} C_VEL
LIN {X 0,Y 376.193,Z 279.801,A -85,B 0,C 180,E1 12662.583,E2 12662.583} C_VEL
LIN {X 0,Y 373.973,Z 275.415,A -85,B 0,C 180,E1 12661.41,E2 12661.41} C_VEL
LIN {X 0,Y 371.66,Z 270.945,A -85,B 0,C 180,E1 12660.155,E2 12660.155} C_VEL
LIN {X 0,Y 369.974,Z 267.854,A -85,B 0,C 180,E1 12659.245,E2 12659.245} C_VEL
LIN {X 0,Y 369.741,Z 266.714,A -85,B 0,C 180,E1 12658.814,E2 12658.814} C_VEL
LIN {X 0,Y 369.735,Z 266.659,A -85,B 0,C 180,E1 12654.643,E2 12654.643} C_VEL
LIN {X 0,Y 369.737,Z 266.657,A -85,B 0,C 180,E1 12650.546,E2 12650.546} C_VEL
LIN {X 0,Y 369.737,Z 266.658,A -85,B 0,C 180,E1 12646.444,E2 12646.444} C_VEL
LIN {X 0,Y 369.741,Z 266.664,A -85,B 0,C 180,E1 12642.324,E2 12642.324} C_VEL
LIN {X 0,Y 369.742,Z 266.677,A -85,B 0,C 180,E1 12638.26,E2 12638.26} C_VEL
LIN {X 0,Y 369.746,Z 266.673,A -85,B 0,C 180,E1 12634.037,E2 12634.037} C_VEL
LIN {X 0,Y 369.751,Z 266.652,A -85,B 0,C 180,E1 12629.837,E2 12629.837} C_VEL
LIN {X 0,Y 369.744,Z 266.651,A -85,B 0,C 180,E1 12625.782,E2 12625.782} C_VEL
LIN {X 0,Y 369.754,Z 266.673,A -85,B 0,C 180,E1 12621.742,E2 12621.742} C_VEL
LIN {X 0,Y 369.746,Z 266.67,A -85,B 0,C 180,E1 12617.628,E2 12617.628} C_VEL
LIN {X 0,Y 369.747,Z 266.646,A -85,B 0,C 180,E1 12613.446,E2 12613.446} C_VEL
LIN {X 0,Y 369.744,Z 266.654,A -85,B 0,C 180,E1 12609.336,E2 12609.336} C_VEL
LIN {X 0,Y 369.747,Z 266.68,A -85,B 0,C 180,E1 12605.274,E2 12605.274} C_VEL
LIN {X 0,Y 369.75,Z 266.668,A -85,B 0,C 180,E1 12601.083,E2 12601.083} C_VEL
LIN {X 0,Y 369.74,Z 266.651,A -85,B 0,C 180,E1 12596.898,E2 12596.898} C_VEL
LIN {X 0,Y 369.752,Z 266.65,A -85,B 0,C 180,E1 12592.853,E2 12592.853} C_VEL
LIN {X 0,Y 369.743,Z 266.66,A -85,B 0,C 180,E1 12588.772,E2 12588.772} C_VEL
LIN {X 0,Y 369.746,Z 266.671,A -85,B 0,C 180,E1 12584.631,E2 12584.631} C_VEL
LIN {X 0,Y 369.744,Z 266.677,A -85,B 0,C 180,E1 12580.571,E2 12580.571} C_VEL
LIN {X 0,Y 369.743,Z 266.675,A -85,B 0,C 180,E1 12576.446,E2 12576.446} C_VEL
LIN {X 0,Y 369.781,Z 266.907,A -85,B 0,C 180,E1 12572.895,E2 12572.895} C_VEL
LIN {X 0,Y 371.266,Z 270.484,A -85,B 0,C 180,E1 12571.881,E2 12571.881} C_VEL
LIN {X 0,Y 372.621,Z 272.287,A -85,B 0,C 180,E1 12571.293,E2 12571.293} C_VEL
LIN {X 0,Y 374.712,Z 276.224,A -85,B 0,C 180,E1 12570.243,E2 12570.243} C_VEL
LIN {X 0,Y 378.406,Z 283.286,A -85,B 0,C 180,E1 12568.454,E2 12568.454} C_VEL
LIN {X 0,Y 382.692,Z 291.151,A -85,B 0,C 180,E1 12566.544,E2 12566.544} C_VEL
LIN {X 0,Y 388.34,Z 302.085,A -85,B 0,C 180,E1 12564.189,E2 12564.189} C_VEL
LIN {X 0,Y 401.024,Z 320.837,A -85,B 0,C 180,E1 12561.577,E2 12561.577} C_VEL
LIN {X 0,Y 412.664,Z 339.401,A -85,B 0,C 180,E1 12559.37,E2 12559.37} C_VEL
LIN {X 0,Y 417.369,Z 347.77,A -85,B 0,C 180,E1 12558.51,E2 12558.51} C_VEL
LIN {X 0,Y 409.526,Z 558.975,A -85,B 0,C 180,E1 12554.563,E2 12554.563} C_VEL
LIN {X 0,Y 407.76,Z 604.249,A -85,B 0,C 180,E1 12553.685,E2 12553.685} C_VEL
LIN {X 0,Y 405.829,Z 626.217,A -85,B 0,C 180,E1 12553.05,E2 12553.05} C_VEL
LIN {X 0,Y 403.352,Z 647.229,A -85,B 0,C 180,E1 12552.202,E2 12552.202} C_VEL
LIN {X 0,Y 400.496,Z 667.597,A -85,B 0,C 180,E1 12551.133,E2 12551.133} C_VEL
LIN {X 0,Y 397.278,Z 686.929,A -85,B 0,C 180,E1 12549.859,E2 12549.859} C_VEL
LIN {X 0,Y 393.622,Z 706.424,A -85,B 0,C 180,E1 12548.287,E2 12548.287} C_VEL
LIN {X 0,Y 389.907,Z 724.845,A -85,B 0,C 180,E1 12546.505,E2 12546.505} C_VEL
LIN {X 0,Y 386.107,Z 742.624,A -85,B 0,C 180,E1 12544.451,E2 12544.451} C_VEL
LIN {X 0,Y 382.371,Z 759.376,A -85,B 0,C 180,E1 12542.147,E2 12542.147} C_VEL
LIN {X 0,Y 378.866,Z 775.252,A -85,B 0,C 180,E1 12539.569,E2 12539.569} C_VEL
LIN {X 0,Y 375.862,Z 789.329,A -85,B 0,C 180,E1 12536.885,E2 12536.885} C_VEL
LIN {X 0,Y 373.308,Z 801.939,A -85,B 0,C 180,E1 12534.022,E2 12534.022} C_VEL
LIN {X 0,Y 371.282,Z 813.251,A -85,B 0,C 180,E1 12530.986,E2 12530.986} C_VEL
LIN {X 0,Y 369.812,Z 822.966,A -85,B 0,C 180,E1 12527.879,E2 12527.879} C_VEL
LIN {X 0,Y 368.866,Z 830.854,A -85,B 0,C 180,E1 12524.76,E2 12524.76} C_VEL
LIN {X 0,Y 368.324,Z 837.556,A -85,B 0,C 180,E1 12521.428,E2 12521.428} C_VEL
LIN {X 0,Y 368.125,Z 842.334,A -85,B 0,C 180,E1 12518.275,E2 12518.275} C_VEL
LIN {X 0,Y 368.1,Z 845.469,A -85,B 0,C 180,E1 12515.141,E2 12515.141} C_VEL
LIN {X 0,Y 368.112,Z 847.214,A -85,B 0,C 180,E1 12512.022,E2 12512.022} C_VEL
LIN {X 0,Y 368.126,Z 847.362,A -85,B 0,C 180,E1 12509.065,E2 12509.065} C_VEL
LIN {X 0,Y 368.101,Z 846.199,A -85,B 0,C 180,E1 12505.949,E2 12505.949} C_VEL
LIN {X 0,Y 368.12,Z 843.405,A -85,B 0,C 180,E1 12502.821,E2 12502.821} C_VEL
LIN {X 0,Y 368.255,Z 838.919,A -85,B 0,C 180,E1 12499.517,E2 12499.517} C_VEL
LIN {X 0,Y 368.644,Z 832.969,A -85,B 0,C 180,E1 12496.35,E2 12496.35} C_VEL
LIN {X 0,Y 369.497,Z 824.892,A -85,B 0,C 180,E1 12493.006,E2 12493.006} C_VEL
LIN {X 0,Y 370.861,Z 815.216,A -85,B 0,C 180,E1 12489.756,E2 12489.756} C_VEL
LIN {X 0,Y 372.791,Z 803.878,A -85,B 0,C 180,E1 12486.611,E2 12486.611} C_VEL
LIN {X 0,Y 375.173,Z 791.486,A -85,B 0,C 180,E1 12483.741,E2 12483.741} C_VEL
LIN {X 0,Y 378.203,Z 777.031,A -85,B 0,C 180,E1 12480.892,E2 12480.892} C_VEL
LIN {X 0,Y 381.602,Z 761.598,A -85,B 0,C 180,E1 12478.307,E2 12478.307} C_VEL
LIN {X 0,Y 385.347,Z 744.575,A -85,B 0,C 180,E1 12475.911,E2 12475.911} C_VEL
LIN {X 0,Y 389.211,Z 726.625,A -85,B 0,C 180,E1 12473.781,E2 12473.781} C_VEL
LIN {X 0,Y 393.058,Z 707.891,A -85,B 0,C 180,E1 12471.911,E2 12471.911} C_VEL
LIN {X 0,Y 396.8,Z 688.429,A -85,B 0,C 180,E1 12470.298,E2 12470.298} C_VEL
LIN {X 0,Y 400.143,Z 668.671,A -85,B 0,C 180,E1 12468.969,E2 12468.969} C_VEL
LIN {X 0,Y 403.333,Z 646.794,A -85,B 0,C 180,E1 12467.792,E2 12467.792} C_VEL
LIN {X 0,Y 405.955,Z 625.22,A -85,B 0,C 180,E1 12466.913,E2 12466.913} C_VEL
LIN {X 0,Y 407.9,Z 603.44,A -85,B 0,C 180,E1 12466.281,E2 12466.281} C_VEL
LIN {X 0,Y 409.511,Z 564.255,A -85,B 0,C 180,E1 12465.509,E2 12465.509} C_VEL
LIN {X 0,Y 417.374,Z 360.556,A -85,B 0,C 180,E1 12461.663,E2 12461.663} C_VEL
LIN {X 0,Y 417.834,Z 346.951,A -85,B 0,C 180,E1 12461.386,E2 12461.386} C_VEL
LIN {X 0,Y 407.87,Z 329.638,A -85,B 0,C 180,E1 12459.346,E2 12459.346} C_VEL
LIN {X 0,Y 397.45,Z 313.492,A -85,B 0,C 180,E1 12457.005,E2 12457.005} C_VEL
LIN {X 0,Y 388.691,Z 300.835,A -85,B 0,C 180,E1 12454.736,E2 12454.736} C_VEL
LIN {X 0,Y 383.687,Z 291.43,A -85,B 0,C 180,E1 12452.115,E2 12452.115} C_VEL
LIN {X 0,Y 381.066,Z 286.676,A -85,B 0,C 180,E1 12450.612,E2 12450.612} C_VEL
LIN {X 0,Y 378.602,Z 282.181,A -85,B 0,C 180,E1 12449.074,E2 12449.074} C_VEL
LIN {X 0,Y 376.524,Z 278.557,A -85,B 0,C 180,E1 12447.692,E2 12447.692} C_VEL
LIN {X 0,Y 375.923,Z 277.341,A -85,B 0,C 180,E1 12447.225,E2 12447.225} C_VEL
LIN {X 0,Y 373.561,Z 273.833,A -85,B 0,C 180,E1 12445.575,E2 12445.575} C_VEL
LIN {X 0,Y 372.651,Z 271.914,A -85,B 0,C 180,E1 12444.745,E2 12444.745} C_VEL
LIN {X 0,Y 370.216,Z 268.543,A -85,B 0,C 180,E1 12442.72,E2 12442.72} C_VEL
LIN {X 0,Y 369.767,Z 266.847,A -85,B 0,C 180,E1 12441.744,E2 12441.744} C_VEL
LIN {X 0,Y 369.735,Z 266.666,A -85,B 0,C 180,E1 12437.631,E2 12437.631} C_VEL
LIN {X 0,Y 369.734,Z 266.668,A -85,B 0,C 180,E1 12433.609,E2 12433.609} C_VEL
LIN {X 0,Y 369.727,Z 266.681,A -85,B 0,C 180,E1 12429.496,E2 12429.496} C_VEL
LIN {X 0,Y 369.724,Z 266.672,A -85,B 0,C 180,E1 12425.432,E2 12425.432} C_VEL
LIN {X 0,Y 369.719,Z 266.668,A -85,B 0,C 180,E1 12421.241,E2 12421.241} C_VEL
LIN {X 0,Y 369.767,Z 267.021,A -85,B 0,C 180,E1 12419.382,E2 12419.382} C_VEL
LIN {X 0,Y 371.759,Z 271.103,A -85,B 0,C 180,E1 12417.072,E2 12417.072} C_VEL
LIN {X 0,Y 373.02,Z 272.49,A -85,B 0,C 180,E1 12416.159,E2 12416.159} C_VEL
LIN {X 0,Y 374.646,Z 276.04,A -85,B 0,C 180,E1 12414.642,E2 12414.642} C_VEL
LIN {X 0,Y 376.001,Z 277.812,A -85,B 0,C 180,E1 12413.742,E2 12413.742} C_VEL
LIN {X 0,Y 377.98,Z 281.649,A -85,B 0,C 180,E1 12412.248,E2 12412.248} C_VEL
LIN {X 0,Y 379.027,Z 283.666,A -85,B 0,C 180,E1 12411.506,E2 12411.506} C_VEL
LIN {X 0,Y 381.485,Z 288.291,A -85,B 0,C 180,E1 12409.888,E2 12409.888} C_VEL
LIN {X 0,Y 384.02,Z 293.385,A -85,B 0,C 180,E1 12408.284,E2 12408.284} C_VEL
LIN {X 0,Y 387.773,Z 300.678,A -85,B 0,C 180,E1 12406.203,E2 12406.203} C_VEL
LIN {X 0,Y 397.402,Z 314.601,A -85,B 0,C 180,E1 12403.71,E2 12403.71} C_VEL
LIN {X 0,Y 406.255,Z 328.356,A -85,B 0,C 180,E1 12401.658,E2 12401.658} C_VEL
LIN {X 0,Y 415.944,Z 344.987,A -85,B 0,C 180,E1 12399.598,E2 12399.598} C_VEL
LIN {X 0,Y 405.398,Z 570.852,A -85,B 0,C 180,E1 12395.106,E2 12395.106} C_VEL
LIN {X 0,Y 403.691,Z 591.655,A -85,B 0,C 180,E1 12394.444,E2 12394.444} C_VEL
LIN {X 0,Y 401.441,Z 611.627,A -85,B 0,C 180,E1 12393.561,E2 12393.561} C_VEL
LIN {X 0,Y 398.697,Z 631.347,A -85,B 0,C 180,E1 12392.425,E2 12392.425} C_VEL
LIN {X 0,Y 395.634,Z 649.899,A -85,B 0,C 180,E1 12391.085,E2 12391.085} C_VEL
LIN {X 0,Y 392.236,Z 667.836,A -85,B 0,C 180,E1 12389.499,E2 12389.499} C_VEL
LIN {X 0,Y 388.525,Z 685.551,A -85,B 0,C 180,E1 12387.577,E2 12387.577} C_VEL
LIN {X 0,Y 384.938,Z 701.345,A -85,B 0,C 180,E1 12385.513,E2 12385.513} C_VEL
LIN {X 0,Y 381.6,Z 715.537,A -85,B 0,C 180,E1 12383.302,E2 12383.302} C_VEL
LIN {X 0,Y 378.432,Z 728.796,A -85,B 0,C 180,E1 12380.844,E2 12380.844} C_VEL
LIN {X 0,Y 375.611,Z 740.77,A -85,B 0,C 180,E1 12378.19,E2 12378.19} C_VEL
LIN {X 0,Y 373.105,Z 751.88,A -85,B 0,C 180,E1 12375.19,E2 12375.19} C_VEL
LIN {X 0,Y 371.203,Z 761.017,A -85,B 0,C 180,E1 12372.122,E2 12372.122} C_VEL
LIN {X 0,Y 369.889,Z 768.289,A -85,B 0,C 180,E1 12369.039,E2 12369.039} C_VEL
LIN {X 0,Y 369.032,Z 774.067,A -85,B 0,C 180,E1 12365.821,E2 12365.821} C_VEL
LIN {X 0,Y 368.579,Z 778.063,A -85,B 0,C 180,E1 12362.674,E2 12362.674} C_VEL
LIN {X 0,Y 368.379,Z 780.475,A -85,B 0,C 180,E1 12359.604,E2 12359.604} C_VEL
LIN {X 0,Y 368.308,Z 781.348,A -85,B 0,C 180,E1 12356.439,E2 12356.439} C_VEL
LIN {X 0,Y 368.323,Z 780.741,A -85,B 0,C 180,E1 12353.351,E2 12353.351} C_VEL
LIN {X 0,Y 368.452,Z 778.763,A -85,B 0,C 180,E1 12350.327,E2 12350.327} C_VEL
LIN {X 0,Y 368.779,Z 775.157,A -85,B 0,C 180,E1 12347.191,E2 12347.191} C_VEL
LIN {X 0,Y 369.408,Z 769.973,A -85,B 0,C 180,E1 12344.101,E2 12344.101} C_VEL
LIN {X 0,Y 370.452,Z 763.223,A -85,B 0,C 180,E1 12341.049,E2 12341.049} C_VEL
LIN {X 0,Y 370.839,Z 761.087,A -85,B 0,C 180,E1 12340.203,E2 12340.203} C_VEL
LIN {X 0,Y 370.42,Z 758.256,A -85,B 0,C 180,E1 12339.087,E2 12339.087} C_VEL
LIN {X 0,Y 366.129,Z 750.274,A -85,B 0,C 180,E1 12336.098,E2 12336.098} C_VEL
LIN {X 0,Y 366.111,Z 747.184,A -85,B 0,C 180,E1 12335.17,E2 12335.17} C_VEL
LIN {X 0,Y 368.72,Z 735.81,A -85,B 0,C 180,E1 12332.333,E2 12332.333} C_VEL
LIN {X 0,Y 371.748,Z 723.067,A -85,B 0,C 180,E1 12329.693,E2 12329.693} C_VEL
LIN {X 0,Y 375.096,Z 708.965,A -85,B 0,C 180,E1 12327.251,E2 12327.251} C_VEL
LIN {X 0,Y 378.57,Z 693.992,A -85,B 0,C 180,E1 12325.077,E2 12325.077} C_VEL
LIN {X 0,Y 382.286,Z 676.85,A -85,B 0,C 180,E1 12323.016,E2 12323.016} C_VEL
LIN {X 0,Y 385.754,Z 659.368,A -85,B 0,C 180,E1 12321.28,E2 12321.28} C_VEL
LIN {X 0,Y 389.009,Z 641.074,A -85,B 0,C 180,E1 12319.786,E2 12319.786} C_VEL
LIN {X 0,Y 391.954,Z 621.958,A -85,B 0,C 180,E1 12318.525,E2 12318.525} C_VEL
LIN {X 0,Y 394.48,Z 602.109,A -85,B 0,C 180,E1 12317.495,E2 12317.495} C_VEL
LIN {X 0,Y 396.546,Z 580.849,A -85,B 0,C 180,E1 12316.677,E2 12316.677} C_VEL
LIN {X 0,Y 397.942,Z 558.877,A -85,B 0,C 180,E1 12316.113,E2 12316.113} C_VEL
LIN {X 0,Y 406.9,Z 346.104,A -85,B 0,C 180,E1 12311.975,E2 12311.975} C_VEL
LIN {X 0,Y 396.106,Z 327.679,A -85,B 0,C 180,E1 12309.88,E2 12309.88} C_VEL
LIN {X 0,Y 385.035,Z 310.577,A -85,B 0,C 180,E1 12307.582,E2 12307.582} C_VEL
LIN {X 0,Y 377.553,Z 299.417,A -85,B 0,C 180,E1 12305.85,E2 12305.85} C_VEL
LIN {X 0,Y 371.271,Z 286.24,A -85,B 0,C 180,E1 12302.582,E2 12302.582} C_VEL
LIN {X 0,Y 366.132,Z 276.517,A -85,B 0,C 180,E1 12299.838,E2 12299.838} C_VEL
LIN {X 0,Y 363.69,Z 271.889,A -85,B 0,C 180,E1 12298.454,E2 12298.454} C_VEL
LIN {X 0,Y 361.954,Z 268.516,A -85,B 0,C 180,E1 12297.404,E2 12297.404} C_VEL
LIN {X 0,Y 361.797,Z 267.693,A -85,B 0,C 180,E1 12297.017,E2 12297.017} C_VEL
LIN {X 0,Y 361.795,Z 267.662,A -85,B 0,C 180,E1 12292.757,E2 12292.757} C_VEL
LIN {X 0,Y 361.797,Z 267.66,A -85,B 0,C 180,E1 12288.665,E2 12288.665} C_VEL
LIN {X 0,Y 361.794,Z 267.653,A -85,B 0,C 180,E1 12284.523,E2 12284.523} C_VEL
LIN {X 0,Y 361.803,Z 267.642,A -85,B 0,C 180,E1 12280.297,E2 12280.297} C_VEL
LIN {X 0,Y 361.796,Z 267.638,A -85,B 0,C 180,E1 12276.203,E2 12276.203} C_VEL
LIN {X 0,Y 361.803,Z 267.649,A -85,B 0,C 180,E1 12272.044,E2 12272.044} C_VEL
LIN {X 0,Y 361.816,Z 267.666,A -85,B 0,C 180,E1 12267.839,E2 12267.839} C_VEL
LIN {X 0,Y 361.81,Z 267.653,A -85,B 0,C 180,E1 12263.621,E2 12263.621} C_VEL
LIN {X 0,Y 361.805,Z 267.634,A -85,B 0,C 180,E1 12259.534,E2 12259.534} C_VEL
LIN {X 0,Y 361.811,Z 267.644,A -85,B 0,C 180,E1 12255.331,E2 12255.331} C_VEL
LIN {X 0,Y 361.806,Z 267.667,A -85,B 0,C 180,E1 12251.152,E2 12251.152} C_VEL
LIN {X 0,Y 361.81,Z 267.648,A -85,B 0,C 180,E1 12246.983,E2 12246.983} C_VEL
LIN {X 0,Y 361.797,Z 267.638,A -85,B 0,C 180,E1 12242.85,E2 12242.85} C_VEL
LIN {X 0,Y 361.799,Z 267.647,A -85,B 0,C 180,E1 12238.732,E2 12238.732} C_VEL
LIN {X 0,Y 361.797,Z 267.665,A -85,B 0,C 180,E1 12234.607,E2 12234.607} C_VEL
LIN {X 0,Y 361.798,Z 267.66,A -85,B 0,C 180,E1 12230.595,E2 12230.595} C_VEL
LIN {X 0,Y 361.794,Z 267.65,A -85,B 0,C 180,E1 12226.413,E2 12226.413} C_VEL
LIN {X 0,Y 361.792,Z 267.648,A -85,B 0,C 180,E1 12222.301,E2 12222.301} C_VEL
LIN {X 0,Y 361.791,Z 267.649,A -85,B 0,C 180,E1 12218.209,E2 12218.209} C_VEL
LIN {X 0,Y 361.843,Z 267.906,A -85,B 0,C 180,E1 12214.705,E2 12214.705} C_VEL
LIN {X 0,Y 363.211,Z 271.317,A -85,B 0,C 180,E1 12213.69,E2 12213.69} C_VEL
LIN {X 0,Y 364.811,Z 273.557,A -85,B 0,C 180,E1 12212.936,E2 12212.936} C_VEL
LIN {X 0,Y 366.841,Z 277.279,A -85,B 0,C 180,E1 12211.866,E2 12211.866} C_VEL
LIN {X 0,Y 370.438,Z 283.945,A -85,B 0,C 180,E1 12210.041,E2 12210.041} C_VEL
LIN {X 0,Y 375.192,Z 292.768,A -85,B 0,C 180,E1 12207.792,E2 12207.792} C_VEL
LIN {X 0,Y 380.003,Z 302.017,A -85,B 0,C 180,E1 12205.685,E2 12205.685} C_VEL
LIN {X 0,Y 391.975,Z 319.256,A -85,B 0,C 180,E1 12203.078,E2 12203.078} C_VEL
LIN {X 0,Y 404.256,Z 338.439,A -85,B 0,C 180,E1 12200.623,E2 12200.623} C_VEL
LIN {X 0,Y 411.584,Z 351.042,A -85,B 0,C 180,E1 12199.234,E2 12199.234} C_VEL
LIN {X 0,Y 403.306,Z 564.39,A -85,B 0,C 180,E1 12195.206,E2 12195.206} C_VEL
LIN {X 0,Y 401.628,Z 604.366,A -85,B 0,C 180,E1 12194.413,E2 12194.413} C_VEL
LIN {X 0,Y 399.632,Z 626.217,A -85,B 0,C 180,E1 12193.774,E2 12193.774} C_VEL
LIN {X 0,Y 396.982,Z 647.66,A -85,B 0,C 180,E1 12192.893,E2 12192.893} C_VEL
LIN {X 0,Y 393.702,Z 669.683,A -85,B 0,C 180,E1 12191.698,E2 12191.698} C_VEL
LIN {X 0,Y 390.349,Z 688.965,A -85,B 0,C 180,E1 12190.392,E2 12190.392} C_VEL
LIN {X 0,Y 386.47,Z 708.47,A -85,B 0,C 180,E1 12188.76,E2 12188.76} C_VEL
LIN {X 0,Y 382.479,Z 727.132,A -85,B 0,C 180,E1 12186.876,E2 12186.876} C_VEL
LIN {X 0,Y 378.523,Z 744.71,A -85,B 0,C 180,E1 12184.764,E2 12184.764} C_VEL
LIN {X 0,Y 374.705,Z 761.038,A -85,B 0,C 180,E1 12182.433,E2 12182.433} C_VEL
LIN {X 0,Y 371.11,Z 776.46,A -85,B 0,C 180,E1 12179.825,E2 12179.825} C_VEL
LIN {X 0,Y 367.855,Z 790.939,A -85,B 0,C 180,E1 12176.933,E2 12176.933} C_VEL
LIN {X 0,Y 365.189,Z 803.735,A -85,B 0,C 180,E1 12173.902,E2 12173.902} C_VEL
LIN {X 0,Y 363.075,Z 815.157,A -85,B 0,C 180,E1 12170.638,E2 12170.638} C_VEL
LIN {X 0,Y 361.624,Z 824.579,A -85,B 0,C 180,E1 12167.372,E2 12167.372} C_VEL
LIN {X 0,Y 360.711,Z 832.424,A -85,B 0,C 180,E1 12164.028,E2 12164.028} C_VEL
LIN {X 0,Y 360.282,Z 838.17,A -85,B 0,C 180,E1 12160.876,E2 12160.876} C_VEL
LIN {X 0,Y 360.121,Z 842.685,A -85,B 0,C 180,E1 12157.496,E2 12157.496} C_VEL
LIN {X 0,Y 360.121,Z 845.35,A -85,B 0,C 180,E1 12154.457,E2 12154.457} C_VEL
LIN {X 0,Y 360.153,Z 846.627,A -85,B 0,C 180,E1 12151.271,E2 12151.271} C_VEL
LIN {X 0,Y 360.151,Z 846.539,A -85,B 0,C 180,E1 12148.407,E2 12148.407} C_VEL
LIN {X 0,Y 360.131,Z 844.996,A -85,B 0,C 180,E1 12145.221,E2 12145.221} C_VEL
LIN {X 0,Y 360.138,Z 842.146,A -85,B 0,C 180,E1 12142.18,E2 12142.18} C_VEL
LIN {X 0,Y 360.318,Z 837.348,A -85,B 0,C 180,E1 12138.798,E2 12138.798} C_VEL
LIN {X 0,Y 360.796,Z 831.218,A -85,B 0,C 180,E1 12135.556,E2 12135.556} C_VEL
LIN {X 0,Y 361.726,Z 823.25,A -85,B 0,C 180,E1 12132.297,E2 12132.297} C_VEL
LIN {X 0,Y 363.314,Z 812.96,A -85,B 0,C 180,E1 12128.866,E2 12128.866} C_VEL
LIN {X 0,Y 365.392,Z 801.776,A -85,B 0,C 180,E1 12125.765,E2 12125.765} C_VEL
LIN {X 0,Y 368.009,Z 789.191,A -85,B 0,C 180,E1 12122.841,E2 12122.841} C_VEL
LIN {X 0,Y 371.108,Z 775.294,A -85,B 0,C 180,E1 12120.102,E2 12120.102} C_VEL
LIN {X 0,Y 374.733,Z 759.668,A -85,B 0,C 180,E1 12117.475,E2 12117.475} C_VEL
LIN {X 0,Y 378.602,Z 743.126,A -85,B 0,C 180,E1 12115.126,E2 12115.126} C_VEL
LIN {X 0,Y 382.523,Z 725.706,A -85,B 0,C 180,E1 12113.044,E2 12113.044} C_VEL
LIN {X 0,Y 386.748,Z 706.11,A -85,B 0,C 180,E1 12111.079,E2 12111.079} C_VEL
LIN {X 0,Y 390.563,Z 687.067,A -85,B 0,C 180,E1 12109.494,E2 12109.494} C_VEL
LIN {X 0,Y 394.093,Z 666.965,A -85,B 0,C 180,E1 12108.143,E2 12108.143} C_VEL
LIN {X 0,Y 397.319,Z 645.619,A -85,B 0,C 180,E1 12107,E2 12107} C_VEL
LIN {X 0,Y 400.032,Z 624.115,A -85,B 0,C 180,E1 12106.127,E2 12106.127} C_VEL
LIN {X 0,Y 402.046,Z 602.271,A -85,B 0,C 180,E1 12105.491,E2 12105.491} C_VEL
LIN {X 0,Y 404.037,Z 554.4,A -85,B 0,C 180,E1 12104.549,E2 12104.549} C_VEL
LIN {X 0,Y 412.243,Z 354.398,A -85,B 0,C 180,E1 12100.724,E2 12100.724} C_VEL
LIN {X 0,Y 412.28,Z 350.292,A -85,B 0,C 180,E1 12100.621,E2 12100.621} C_VEL
LIN {X 0,Y 403.327,Z 334.661,A -85,B 0,C 180,E1 12098.707,E2 12098.707} C_VEL
LIN {X 0,Y 393.837,Z 319.712,A -85,B 0,C 180,E1 12096.492,E2 12096.492} C_VEL
LIN {X 0,Y 384.564,Z 306.547,A -85,B 0,C 180,E1 12094.077,E2 12094.077} C_VEL
LIN {X 0,Y 380.399,Z 300.711,A -85,B 0,C 180,E1 12092.784,E2 12092.784} C_VEL
LIN {X 0,Y 378.221,Z 296.63,A -85,B 0,C 180,E1 12091.563,E2 12091.563} C_VEL
LIN {X 0,Y 376.212,Z 292.794,A -85,B 0,C 180,E1 12090.33,E2 12090.33} C_VEL
LIN {X 0,Y 374.075,Z 288.713,A -85,B 0,C 180,E1 12088.934,E2 12088.934} C_VEL
LIN {X 0,Y 371.827,Z 284.696,A -85,B 0,C 180,E1 12087.377,E2 12087.377} C_VEL
LIN {X 0,Y 368.92,Z 279.865,A -85,B 0,C 180,E1 12085.184,E2 12085.184} C_VEL
